dipar.Vn1_AVOM_ON(mdl_value := MODULE_UCP1_A2_DI3.VALUE.2, mdl_flt := MODULE_UCP1_A2_DI3.HwError); //Вентилятор АВОМД+Н+У №1 включен
dipar.Vn2_AVOM_ON(mdl_value := MODULE_UCP1_A2_DI3.VALUE.3, mdl_flt := MODULE_UCP1_A2_DI3.HwError); //Вентилятор АВОМД+Н+У №2 включен
dipar.VV_VOU_ON(mdl_value := MODULE_UCP1_A2_DI3.VALUE.4, mdl_flt := MODULE_UCP1_A2_DI3.HwError); //Вентилятор ВОУ включен
dipar.VVN_ON(mdl_value := MODULE_UCP1_A2_DI3.VALUE.5, mdl_flt := MODULE_UCP1_A2_DI3.HwError); //Вытяжной вентилятор нагнетателя ВВН включен
dipar.TRKready(mdl_value := MODULE_UCP1_A2_DI3.VALUE.8, mdl_flt := MODULE_UCP1_A2_DI3.HwError); //ТРК: готовность
dipar.TRKalr(mdl_value := MODULE_UCP1_A2_DI3.VALUE.9, mdl_flt := MODULE_UCP1_A2_DI3.HwError); //ТРК: авария
dipar.Ptg_inDG_Pn(mdl_value := MODULE_UCP1_A2_DI3.VALUE.17, mdl_flt := MODULE_UCP1_A2_DI3.HwError); //Давление газа перед дозатором газа Предупредительное
dipar.Vn3_AVOM_ON(mdl_value := MODULE_UCP1_A2_DI3.VALUE.21, mdl_flt := MODULE_UCP1_A2_DI3.HwError); //Вентилятор АВОМД+Н+У №3 включен
dipar.Vn4_AVOM_ON(mdl_value := MODULE_UCP1_A2_DI3.VALUE.22, mdl_flt := MODULE_UCP1_A2_DI3.HwError); //Вентилятор АВОМД+Н+У №4 включен
dipar.Ptg_inDG_An(mdl_value := MODULE_UCP1_A2_DI3.VALUE.23, mdl_flt := MODULE_UCP1_A2_DI3.HwError); //Давление газа перед дозатором газа Аварийное
dipar.Fuse_AO_UCP1(mdl_value := MODULE_UCP1_A2_DI4.VALUE.16, mdl_flt := MODULE_UCP1_A2_DI4.HwError); //диаг. Предохранитель UCP1-XTFU1:1 питания модулей AO исправен
dipar.Fuse_DO_UCP1(mdl_value := MODULE_UCP1_A2_DI4.VALUE.17, mdl_flt := MODULE_UCP1_A2_DI4.HwError); //диаг. Предохранитель UCP1-XTFU1:2 питания модулей DO исправен
dipar.Fuse_Air_UCP1(mdl_value := MODULE_UCP1_A2_DI4.VALUE.18, mdl_flt := MODULE_UCP1_A2_DI4.HwError); //диаг. Предохранитель UCP1--XTFU6:1 питания датчиков температуры и влажности
dipar.AO_PRU_1_ai(mdl_value := MODULE_UE1_A1_DI1.CH01.VALUE, mdl_flt := MODULE_UE1_A1_DI1.CH01.STATUS.0 OR MODULE_UE1_A1_DI1.HwError); //Кнопка АО на ПРУ сигнал 1 (НР)
dipar.AO_PRU_1(mdl_value := dipar.AO_PRU_1_ai.value, mdl_hwError := dipar.AO_PRU_1_ai.flt, mdl_sc := dipar.AO_PRU_1_ai.sc, mdl_brk := dipar.AO_PRU_1_ai.brk); //Кнопка АО на ПРУ сигнал 1 (НР)

dipar.Kr1_off_ai(mdl_value := MODULE_UE1_A1_DI1.CH02.VALUE, mdl_flt := MODULE_UE1_A1_DI1.CH02.STATUS.0 OR MODULE_UE1_A1_DI1.HwError); //Кран 1 закрыт
dipar.Kr1_off(mdl_value := dipar.Kr1_off_ai.value, mdl_hwError := dipar.Kr1_off_ai.flt, mdl_sc := dipar.Kr1_off_ai.sc, mdl_brk := dipar.Kr1_off_ai.brk); //Кран 1 закрыт

dipar.Kr2_off_ai(mdl_value := MODULE_UE1_A1_DI1.CH03.VALUE, mdl_flt := MODULE_UE1_A1_DI1.CH03.STATUS.0 OR MODULE_UE1_A1_DI1.HwError); //Кран 2 закрыт
dipar.Kr2_off(mdl_value := dipar.Kr2_off_ai.value, mdl_hwError := dipar.Kr2_off_ai.flt, mdl_sc := dipar.Kr2_off_ai.sc, mdl_brk := dipar.Kr2_off_ai.brk); //Кран 2 закрыт

dipar.Kr4_off_ai(mdl_value := MODULE_UE1_A1_DI1.CH04.VALUE, mdl_flt := MODULE_UE1_A1_DI1.CH04.STATUS.0 OR MODULE_UE1_A1_DI1.HwError); //Кран 4 закрыт
dipar.Kr4_off(mdl_value := dipar.Kr4_off_ai.value, mdl_hwError := dipar.Kr4_off_ai.flt, mdl_sc := dipar.Kr4_off_ai.sc, mdl_brk := dipar.Kr4_off_ai.brk); //Кран 4 закрыт

dipar.Kr5_off_ai(mdl_value := MODULE_UE1_A1_DI1.CH05.VALUE, mdl_flt := MODULE_UE1_A1_DI1.CH05.STATUS.0 OR MODULE_UE1_A1_DI1.HwError); //Кран 5 закрыт
dipar.Kr5_off(mdl_value := dipar.Kr5_off_ai.value, mdl_hwError := dipar.Kr5_off_ai.flt, mdl_sc := dipar.Kr5_off_ai.sc, mdl_brk := dipar.Kr5_off_ai.brk); //Кран 5 закрыт

dipar.Kr6_off_ai(mdl_value := MODULE_UE1_A1_DI1.CH06.VALUE, mdl_flt := MODULE_UE1_A1_DI1.CH06.STATUS.0 OR MODULE_UE1_A1_DI1.HwError); //Кран 6 закрыт
dipar.Kr6_off(mdl_value := dipar.Kr6_off_ai.value, mdl_hwError := dipar.Kr6_off_ai.flt, mdl_sc := dipar.Kr6_off_ai.sc, mdl_brk := dipar.Kr6_off_ai.brk); //Кран 6 закрыт

dipar.Kr12_off_ai(mdl_value := MODULE_UE1_A1_DI1.CH07.VALUE, mdl_flt := MODULE_UE1_A1_DI1.CH07.STATUS.0 OR MODULE_UE1_A1_DI1.HwError); //Кран 12 закрыт (т.г.)
dipar.Kr12_off(mdl_value := dipar.Kr12_off_ai.value, mdl_hwError := dipar.Kr12_off_ai.flt, mdl_sc := dipar.Kr12_off_ai.sc, mdl_brk := dipar.Kr12_off_ai.brk); //Кран 12 закрыт (т.г.)

dipar.Kr9_off_ai(mdl_value := MODULE_UE1_A1_DI1.CH08.VALUE, mdl_flt := MODULE_UE1_A1_DI1.CH08.STATUS.0 OR MODULE_UE1_A1_DI1.HwError); //Кран 9 закрыт (т.газ. свеча.)
dipar.Kr9_off(mdl_value := dipar.Kr9_off_ai.value, mdl_hwError := dipar.Kr9_off_ai.flt, mdl_sc := dipar.Kr9_off_ai.sc, mdl_brk := dipar.Kr9_off_ai.brk); //Кран 9 закрыт (т.газ. свеча.)

dipar.Kr11_off_ai(mdl_value := MODULE_UE1_A1_DI1.CH09.VALUE, mdl_flt := MODULE_UE1_A1_DI1.CH09.STATUS.0 OR MODULE_UE1_A1_DI1.HwError); //Кран 11 закрыт (п.г.)
dipar.Kr11_off(mdl_value := dipar.Kr11_off_ai.value, mdl_hwError := dipar.Kr11_off_ai.flt, mdl_sc := dipar.Kr11_off_ai.sc, mdl_brk := dipar.Kr11_off_ai.brk); //Кран 11 закрыт (п.г.)

dipar.Kr10_off_ai(mdl_value := MODULE_UE1_A1_DI1.CH10.VALUE, mdl_flt := MODULE_UE1_A1_DI1.CH10.STATUS.0 OR MODULE_UE1_A1_DI1.HwError); //Кран 10 закрыт (п.газ. свеча.)
dipar.Kr10_off(mdl_value := dipar.Kr10_off_ai.value, mdl_hwError := dipar.Kr10_off_ai.flt, mdl_sc := dipar.Kr10_off_ai.sc, mdl_brk := dipar.Kr10_off_ai.brk); //Кран 10 закрыт (п.газ. свеча.)

dipar.KPV1_off_ai(mdl_value := MODULE_UE1_A1_DI1.CH11.VALUE, mdl_flt := MODULE_UE1_A1_DI1.CH11.STATUS.0 OR MODULE_UE1_A1_DI1.HwError); //КПВ-1 закрыт
dipar.KPV1_off(mdl_value := dipar.KPV1_off_ai.value, mdl_hwError := dipar.KPV1_off_ai.flt, mdl_sc := dipar.KPV1_off_ai.sc, mdl_brk := dipar.KPV1_off_ai.brk); //КПВ-1 закрыт

dipar.KPV2_off_ai(mdl_value := MODULE_UE1_A1_DI1.CH12.VALUE, mdl_flt := MODULE_UE1_A1_DI1.CH12.STATUS.0 OR MODULE_UE1_A1_DI1.HwError); //КПВ-2 закрыт
dipar.KPV2_off(mdl_value := dipar.KPV2_off_ai.value, mdl_hwError := dipar.KPV2_off_ai.flt, mdl_sc := dipar.KPV2_off_ai.sc, mdl_brk := dipar.KPV2_off_ai.brk); //КПВ-2 закрыт

dipar.KPV3_off_ai(mdl_value := MODULE_UE1_A1_DI1.CH13.VALUE, mdl_flt := MODULE_UE1_A1_DI1.CH13.STATUS.0 OR MODULE_UE1_A1_DI1.HwError); //КПВ-3 закрыт
dipar.KPV3_off(mdl_value := dipar.KPV3_off_ai.value, mdl_hwError := dipar.KPV3_off_ai.flt, mdl_sc := dipar.KPV3_off_ai.sc, mdl_brk := dipar.KPV3_off_ai.brk); //КПВ-3 закрыт

dipar.KPV4_off_ai(mdl_value := MODULE_UE1_A1_DI1.CH14.VALUE, mdl_flt := MODULE_UE1_A1_DI1.CH14.STATUS.0 OR MODULE_UE1_A1_DI1.HwError); //КПВ-4 закрыт
dipar.KPV4_off(mdl_value := dipar.KPV4_off_ai.value, mdl_hwError := dipar.KPV4_off_ai.flt, mdl_sc := dipar.KPV4_off_ai.sc, mdl_brk := dipar.KPV4_off_ai.brk); //КПВ-4 закрыт

dipar.KPV5_off_ai(mdl_value := MODULE_UE1_A1_DI1.CH15.VALUE, mdl_flt := MODULE_UE1_A1_DI1.CH15.STATUS.0 OR MODULE_UE1_A1_DI1.HwError); //КПВ-5 закрыт
dipar.KPV5_off(mdl_value := dipar.KPV5_off_ai.value, mdl_hwError := dipar.KPV5_off_ai.flt, mdl_sc := dipar.KPV5_off_ai.sc, mdl_brk := dipar.KPV5_off_ai.brk); //КПВ-5 закрыт

dipar.SK_off_ai(mdl_value := MODULE_UE1_A1_DI1.CH16.VALUE, mdl_flt := MODULE_UE1_A1_DI1.CH16.STATUS.0 OR MODULE_UE1_A1_DI1.HwError); //СК закрыт
dipar.SK_off(mdl_value := dipar.SK_off_ai.value, mdl_hwError := dipar.SK_off_ai.flt, mdl_sc := dipar.SK_off_ai.sc, mdl_brk := dipar.SK_off_ai.brk); //СК закрыт

dipar.AO_PRU_2_ai(mdl_value := MODULE_UE1_A1_DI2.CH01.VALUE, mdl_flt := MODULE_UE1_A1_DI2.CH01.STATUS.0 OR MODULE_UE1_A1_DI2.HwError); //Кнопка АО на ПРУ сигнал 2 (НЗ)
dipar.AO_PRU_2(mdl_value := dipar.AO_PRU_2_ai.value, mdl_hwError := dipar.AO_PRU_2_ai.flt, mdl_sc := dipar.AO_PRU_2_ai.sc, mdl_brk := dipar.AO_PRU_2_ai.brk); //Кнопка АО на ПРУ сигнал 2 (НЗ)

dipar.Kr1_ON_ai(mdl_value := MODULE_UE1_A1_DI2.CH02.VALUE, mdl_flt := MODULE_UE1_A1_DI2.CH02.STATUS.0 OR MODULE_UE1_A1_DI2.HwError); //Кран 1 открыт
dipar.Kr1_ON(mdl_value := dipar.Kr1_ON_ai.value, mdl_hwError := dipar.Kr1_ON_ai.flt, mdl_sc := dipar.Kr1_ON_ai.sc, mdl_brk := dipar.Kr1_ON_ai.brk); //Кран 1 открыт

dipar.Kr2_ON_ai(mdl_value := MODULE_UE1_A1_DI2.CH03.VALUE, mdl_flt := MODULE_UE1_A1_DI2.CH03.STATUS.0 OR MODULE_UE1_A1_DI2.HwError); //Кран 2 открыт
dipar.Kr2_ON(mdl_value := dipar.Kr2_ON_ai.value, mdl_hwError := dipar.Kr2_ON_ai.flt, mdl_sc := dipar.Kr2_ON_ai.sc, mdl_brk := dipar.Kr2_ON_ai.brk); //Кран 2 открыт

dipar.Kr4_ON_ai(mdl_value := MODULE_UE1_A1_DI2.CH04.VALUE, mdl_flt := MODULE_UE1_A1_DI2.CH04.STATUS.0 OR MODULE_UE1_A1_DI2.HwError); //Кран 4 открыт
dipar.Kr4_ON(mdl_value := dipar.Kr4_ON_ai.value, mdl_hwError := dipar.Kr4_ON_ai.flt, mdl_sc := dipar.Kr4_ON_ai.sc, mdl_brk := dipar.Kr4_ON_ai.brk); //Кран 4 открыт

dipar.Kr5_ON_ai(mdl_value := MODULE_UE1_A1_DI2.CH05.VALUE, mdl_flt := MODULE_UE1_A1_DI2.CH05.STATUS.0 OR MODULE_UE1_A1_DI2.HwError); //Кран 5 открыт
dipar.Kr5_ON(mdl_value := dipar.Kr5_ON_ai.value, mdl_hwError := dipar.Kr5_ON_ai.flt, mdl_sc := dipar.Kr5_ON_ai.sc, mdl_brk := dipar.Kr5_ON_ai.brk); //Кран 5 открыт

dipar.Kr6_ON_ai(mdl_value := MODULE_UE1_A1_DI2.CH06.VALUE, mdl_flt := MODULE_UE1_A1_DI2.CH06.STATUS.0 OR MODULE_UE1_A1_DI2.HwError); //Кран 6 открыт
dipar.Kr6_ON(mdl_value := dipar.Kr6_ON_ai.value, mdl_hwError := dipar.Kr6_ON_ai.flt, mdl_sc := dipar.Kr6_ON_ai.sc, mdl_brk := dipar.Kr6_ON_ai.brk); //Кран 6 открыт

dipar.Kr12_ON_ai(mdl_value := MODULE_UE1_A1_DI2.CH07.VALUE, mdl_flt := MODULE_UE1_A1_DI2.CH07.STATUS.0 OR MODULE_UE1_A1_DI2.HwError); //Кран 12 открыт (т.г.)
dipar.Kr12_ON(mdl_value := dipar.Kr12_ON_ai.value, mdl_hwError := dipar.Kr12_ON_ai.flt, mdl_sc := dipar.Kr12_ON_ai.sc, mdl_brk := dipar.Kr12_ON_ai.brk); //Кран 12 открыт (т.г.)

dipar.Kr9_ON_ai(mdl_value := MODULE_UE1_A1_DI2.CH08.VALUE, mdl_flt := MODULE_UE1_A1_DI2.CH08.STATUS.0 OR MODULE_UE1_A1_DI2.HwError); //Кран 9 открыт (т.газ. свеча.)
dipar.Kr9_ON(mdl_value := dipar.Kr9_ON_ai.value, mdl_hwError := dipar.Kr9_ON_ai.flt, mdl_sc := dipar.Kr9_ON_ai.sc, mdl_brk := dipar.Kr9_ON_ai.brk); //Кран 9 открыт (т.газ. свеча.)

dipar.Kr11_ON_ai(mdl_value := MODULE_UE1_A1_DI2.CH09.VALUE, mdl_flt := MODULE_UE1_A1_DI2.CH09.STATUS.0 OR MODULE_UE1_A1_DI2.HwError); //Кран 11 открыт (п.г.)
dipar.Kr11_ON(mdl_value := dipar.Kr11_ON_ai.value, mdl_hwError := dipar.Kr11_ON_ai.flt, mdl_sc := dipar.Kr11_ON_ai.sc, mdl_brk := dipar.Kr11_ON_ai.brk); //Кран 11 открыт (п.г.)

dipar.Kr10_ON_ai(mdl_value := MODULE_UE1_A1_DI2.CH10.VALUE, mdl_flt := MODULE_UE1_A1_DI2.CH10.STATUS.0 OR MODULE_UE1_A1_DI2.HwError); //Кран 10 открыт (п.газ. свеча.)
dipar.Kr10_ON(mdl_value := dipar.Kr10_ON_ai.value, mdl_hwError := dipar.Kr10_ON_ai.flt, mdl_sc := dipar.Kr10_ON_ai.sc, mdl_brk := dipar.Kr10_ON_ai.brk); //Кран 10 открыт (п.газ. свеча.)

dipar.KPV1_ON_ai(mdl_value := MODULE_UE1_A1_DI2.CH11.VALUE, mdl_flt := MODULE_UE1_A1_DI2.CH11.STATUS.0 OR MODULE_UE1_A1_DI2.HwError); //КПВ-1 открыт
dipar.KPV1_ON(mdl_value := dipar.KPV1_ON_ai.value, mdl_hwError := dipar.KPV1_ON_ai.flt, mdl_sc := dipar.KPV1_ON_ai.sc, mdl_brk := dipar.KPV1_ON_ai.brk); //КПВ-1 открыт

dipar.KPV2_ON_ai(mdl_value := MODULE_UE1_A1_DI2.CH12.VALUE, mdl_flt := MODULE_UE1_A1_DI2.CH12.STATUS.0 OR MODULE_UE1_A1_DI2.HwError); //КПВ-2 открыт
dipar.KPV2_ON(mdl_value := dipar.KPV2_ON_ai.value, mdl_hwError := dipar.KPV2_ON_ai.flt, mdl_sc := dipar.KPV2_ON_ai.sc, mdl_brk := dipar.KPV2_ON_ai.brk); //КПВ-2 открыт

dipar.KPV3_ON_ai(mdl_value := MODULE_UE1_A1_DI2.CH13.VALUE, mdl_flt := MODULE_UE1_A1_DI2.CH13.STATUS.0 OR MODULE_UE1_A1_DI2.HwError); //КПВ-3 открыт
dipar.KPV3_ON(mdl_value := dipar.KPV3_ON_ai.value, mdl_hwError := dipar.KPV3_ON_ai.flt, mdl_sc := dipar.KPV3_ON_ai.sc, mdl_brk := dipar.KPV3_ON_ai.brk); //КПВ-3 открыт

dipar.KPV4_ON_ai(mdl_value := MODULE_UE1_A1_DI2.CH14.VALUE, mdl_flt := MODULE_UE1_A1_DI2.CH14.STATUS.0 OR MODULE_UE1_A1_DI2.HwError); //КПВ-4 открыт
dipar.KPV4_ON(mdl_value := dipar.KPV4_ON_ai.value, mdl_hwError := dipar.KPV4_ON_ai.flt, mdl_sc := dipar.KPV4_ON_ai.sc, mdl_brk := dipar.KPV4_ON_ai.brk); //КПВ-4 открыт

dipar.KPV5_ON_ai(mdl_value := MODULE_UE1_A1_DI2.CH15.VALUE, mdl_flt := MODULE_UE1_A1_DI2.CH15.STATUS.0 OR MODULE_UE1_A1_DI2.HwError); //КПВ-5 открыт
dipar.KPV5_ON(mdl_value := dipar.KPV5_ON_ai.value, mdl_hwError := dipar.KPV5_ON_ai.flt, mdl_sc := dipar.KPV5_ON_ai.sc, mdl_brk := dipar.KPV5_ON_ai.brk); //КПВ-5 открыт

dipar.SK_ON_ai(mdl_value := MODULE_UE1_A1_DI2.CH16.VALUE, mdl_flt := MODULE_UE1_A1_DI2.CH16.STATUS.0 OR MODULE_UE1_A1_DI2.HwError); //СК открыт
dipar.SK_ON(mdl_value := dipar.SK_ON_ai.value, mdl_hwError := dipar.SK_ON_ai.flt, mdl_sc := dipar.SK_ON_ai.sc, mdl_brk := dipar.SK_ON_ai.brk); //СК открыт

dipar.PNS_ON_ai(mdl_value := MODULE_UE1_A1_DI3.CH01.VALUE, mdl_flt := MODULE_UE1_A1_DI3.CH01.STATUS.0 OR MODULE_UE1_A1_DI3.HwError); //Пусковой насос смазки включен
dipar.PNS_ON(mdl_value := dipar.PNS_ON_ai.value, mdl_hwError := dipar.PNS_ON_ai.flt, mdl_sc := dipar.PNS_ON_ai.sc, mdl_brk := dipar.PNS_ON_ai.brk); //Пусковой насос смазки включен

dipar.PNU_ON_ai(mdl_value := MODULE_UE1_A1_DI3.CH02.VALUE, mdl_flt := MODULE_UE1_A1_DI3.CH02.STATUS.0 OR MODULE_UE1_A1_DI3.HwError); //Пусковой насос уплотнения включен
dipar.PNU_ON(mdl_value := dipar.PNU_ON_ai.value, mdl_hwError := dipar.PNU_ON_ai.flt, mdl_sc := dipar.PNU_ON_ai.sc, mdl_brk := dipar.PNU_ON_ai.brk); //Пусковой насос уплотнения включен

dipar.Vs_D_Pv(mdl_value := MODULE_UE1_A1_DI4.VALUE.8, mdl_flt := MODULE_UE1_A1_DI4.HwError); //Повышенная вибрация двигателя
dipar.Vs_D_Av(mdl_value := MODULE_UE1_A1_DI4.VALUE.9, mdl_flt := MODULE_UE1_A1_DI4.HwError); //Опасная вибрация двигателя
dipar.Zs_Nl(mdl_value := MODULE_UE1_A1_DI4.VALUE.17, mdl_flt := MODULE_UE1_A1_DI4.HwError); //Осевой сдвиг ротора Н Аварийный
dipar.Pg_outKR1(mdl_value := MODULE_UE1_A1_DI4.VALUE.19, mdl_flt := MODULE_UE1_A1_DI4.HwError); //Давление газа после крана 1
dipar.Pm_N_Pn(mdl_value := MODULE_UE1_A1_DI4.VALUE.22, mdl_flt := MODULE_UE1_A1_DI4.HwError); //Давление масла смазки Н предупредительная
dipar.Exh_VOU(mdl_value := MODULE_UE1_A1_DI4.VALUE.23, mdl_flt := MODULE_UE1_A1_DI4.HwError); //Разрежение в ВОУ
dipar.Pg_InKR13(mdl_value := MODULE_UE1_A1_DI4.VALUE.24, mdl_flt := MODULE_UE1_A1_DI4.HwError); //Давление газа до крана 13 (воздушного стартера)
dipar.Pm_Starter_Av(mdl_value := MODULE_UE1_A1_DI4.VALUE.25, mdl_flt := MODULE_UE1_A1_DI4.HwError); //Давление масла смазки воздушного стартера высокий уровень
dipar.Pm_Starter_An(mdl_value := MODULE_UE1_A1_DI4.VALUE.26, mdl_flt := MODULE_UE1_A1_DI4.HwError); //Давление масла смазки воздушного стартера низкий уровень
dipar.EAO_PRU_1(mdl_value := MODULE_UE1_A1_DI4.VALUE.28, mdl_flt := MODULE_UE1_A1_DI4.HwError); //Кнопка ЭАО на ПРУ нажата сигнал 1 (НР)
dipar.EAO_PRU_2(mdl_value := MODULE_UE1_A1_DI4.VALUE.29, mdl_flt := MODULE_UE1_A1_DI4.HwError); //Кнопка ЭАО на ПРУ нажата сигнал 2 (НЗ)
dipar.EAO_PRU_3(mdl_value := MODULE_UE1_A1_DI4.VALUE.30, mdl_flt := MODULE_UE1_A1_DI4.HwError); //Кнопка ЭАО на ПРУ нажата сигнал 3 (НЗ)
dipar.BEAO(mdl_value := MODULE_UE1_A1_DI4.VALUE.31, mdl_flt := MODULE_UE1_A1_DI4.HwError); //БЭАО сработал
dipar.Kr13_ON(mdl_value := MODULE_UE1_A1_DI5.VALUE.0, mdl_flt := MODULE_UE1_A1_DI5.HwError); //Заслонка ВC (кран 13) открыта
dipar.BZA_alr(mdl_value := MODULE_UE1_A1_DI5.VALUE.1, mdl_flt := MODULE_UE1_A1_DI5.HwError); //БЗА. Авария
dipar.BZA_ready_1(mdl_value := MODULE_UE1_A1_DI5.VALUE.2, mdl_flt := MODULE_UE1_A1_DI5.HwError); //БЗА. Готовность 1
dipar.BZA_ready_2(mdl_value := MODULE_UE1_A1_DI5.VALUE.3, mdl_flt := MODULE_UE1_A1_DI5.HwError); //БЗА. Готовность 2
dipar.U_CC_cntrl(mdl_value := MODULE_UE1_A1_DI5.VALUE.24, mdl_flt := MODULE_UE1_A1_DI5.HwError); //Контроль питания СС
dipar.Chip_outD(mdl_value := MODULE_UE1_A1_DI5.VALUE.25, mdl_flt := MODULE_UE1_A1_DI5.HwError); //Стружка в масле на выходе Д
dipar.Ace_alr(mdl_value := MODULE_UE1_A1_DI5.VALUE.26, mdl_flt := MODULE_UE1_A1_DI5.HwError); //Сигнализатор обледенения
dipar.kcdo_Kr1_off(mdl_value := MODULE_UE1_A1_DI6.VALUE.0, mdl_flt := MODULE_UE1_A1_DI6.HwError); //диаг. Кран 1 закрыть
dipar.kcdo_Kr1m_ON(mdl_value := MODULE_UE1_A1_DI6.VALUE.1, mdl_flt := MODULE_UE1_A1_DI6.HwError); //диаг. Кран 1 смазка
dipar.kcdo_Kr2_off(mdl_value := MODULE_UE1_A1_DI6.VALUE.2, mdl_flt := MODULE_UE1_A1_DI6.HwError); //диаг. Кран 2 закрыть
dipar.kcdo_Kr2m_ON(mdl_value := MODULE_UE1_A1_DI6.VALUE.3, mdl_flt := MODULE_UE1_A1_DI6.HwError); //диаг. Кран 2 смазка
dipar.kcdo_Kr4_off(mdl_value := MODULE_UE1_A1_DI6.VALUE.4, mdl_flt := MODULE_UE1_A1_DI6.HwError); //диаг. Кран 4 закрыть
dipar.kcdo_Kr4m_ON(mdl_value := MODULE_UE1_A1_DI6.VALUE.5, mdl_flt := MODULE_UE1_A1_DI6.HwError); //диаг. Кран 4 смазка
dipar.kcdo_Kr5_ON(mdl_value := MODULE_UE1_A1_DI6.VALUE.6, mdl_flt := MODULE_UE1_A1_DI6.HwError); //диаг. Кран 5 открыть
dipar.kcdo_Kr5m_ON(mdl_value := MODULE_UE1_A1_DI6.VALUE.7, mdl_flt := MODULE_UE1_A1_DI6.HwError); //диаг. Кран 5 смазка
dipar.kcdo_Kr6_off(mdl_value := MODULE_UE1_A1_DI6.VALUE.8, mdl_flt := MODULE_UE1_A1_DI6.HwError); //диаг. Кран 6 закрыть
dipar.kcdo_Kr6m_ON(mdl_value := MODULE_UE1_A1_DI6.VALUE.9, mdl_flt := MODULE_UE1_A1_DI6.HwError); //диаг. Кран 6 смазка
dipar.kcdo_KR12_off(mdl_value := MODULE_UE1_A1_DI6.VALUE.10, mdl_flt := MODULE_UE1_A1_DI6.HwError); //диаг. Кран 12 закрыть (т.г.)
dipar.kcdo_KR12m_ON(mdl_value := MODULE_UE1_A1_DI6.VALUE.11, mdl_flt := MODULE_UE1_A1_DI6.HwError); //диаг. Кран 12 смазка
dipar.kcdo_KR9m_ON(mdl_value := MODULE_UE1_A1_DI6.VALUE.13, mdl_flt := MODULE_UE1_A1_DI6.HwError); //диаг. Кран 9 смазка
dipar.kcdo_Kr11_ON(mdl_value := MODULE_UE1_A1_DI6.VALUE.14, mdl_flt := MODULE_UE1_A1_DI6.HwError); //диаг. Кран 11 открыть (п.г.)
dipar.kcdo_Kr11m_ON(mdl_value := MODULE_UE1_A1_DI6.VALUE.15, mdl_flt := MODULE_UE1_A1_DI6.HwError); //диаг. Кран 11 смазка
dipar.kcdo_Kr10m_ON(mdl_value := MODULE_UE1_A1_DI6.VALUE.17, mdl_flt := MODULE_UE1_A1_DI6.HwError); //диаг. Кран 10 смазка
dipar.kcdo_KPV15_ON(mdl_value := MODULE_UE1_A1_DI6.VALUE.18, mdl_flt := MODULE_UE1_A1_DI6.HwError); //диаг. Включение КПВ 1,5
dipar.kcdo_KPV23_off(mdl_value := MODULE_UE1_A1_DI6.VALUE.19, mdl_flt := MODULE_UE1_A1_DI6.HwError); //диаг. Включение КПВ 2,3
dipar.kcdo_KPV4_off(mdl_value := MODULE_UE1_A1_DI6.VALUE.20, mdl_flt := MODULE_UE1_A1_DI6.HwError); //диаг. Включение КПВ 4
dipar.kcdo_SK_ON(mdl_value := MODULE_UE1_A1_DI6.VALUE.21, mdl_flt := MODULE_UE1_A1_DI6.HwError); //диаг. Стопорный клапан открыть
dipar.kcdo_Kr1_ON(mdl_value := MODULE_UE1_A1_DI7.VALUE.0, mdl_flt := MODULE_UE1_A1_DI7.HwError); //диаг. Кран 1 открыть
dipar.kcdo_Kr2_ON(mdl_value := MODULE_UE1_A1_DI7.VALUE.1, mdl_flt := MODULE_UE1_A1_DI7.HwError); //диаг. Кран 2 открыть
dipar.kcdo_Kr4_ON(mdl_value := MODULE_UE1_A1_DI7.VALUE.2, mdl_flt := MODULE_UE1_A1_DI7.HwError); //диаг. Кран 4 открыть
dipar.kcdo_Kr5_off(mdl_value := MODULE_UE1_A1_DI7.VALUE.3, mdl_flt := MODULE_UE1_A1_DI7.HwError); //диаг. Кран 5 закрыть
dipar.kcdo_Kr6_ON(mdl_value := MODULE_UE1_A1_DI7.VALUE.4, mdl_flt := MODULE_UE1_A1_DI7.HwError); //диаг. Кран 6 открыть
dipar.kcdo_Kr12_ON(mdl_value := MODULE_UE1_A1_DI7.VALUE.5, mdl_flt := MODULE_UE1_A1_DI7.HwError); //диаг. Кран 12 открыть (т.г.)
dipar.kcdo_Kr11_off(mdl_value := MODULE_UE1_A1_DI7.VALUE.7, mdl_flt := MODULE_UE1_A1_DI7.HwError); //диаг. Кран 11 закрыть (п.г.)
dipar.kcdo_Sound_ON(mdl_value := MODULE_UE1_A1_DI7.VALUE.10, mdl_flt := MODULE_UE1_A1_DI7.HwError); //диаг. ЗВУКОВУЮ СИГНАЛИЗАЦИЮ в ГЩУ ВКЛЮЧИТЬ
dipar.kcdo_VNA_ON(mdl_value := MODULE_UE1_A1_DI7.VALUE.15, mdl_flt := MODULE_UE1_A1_DI7.HwError); //диаг. Эл. магнит управления ВНА включить
dipar.Fuse_DO_UE1(mdl_value := MODULE_UE1_A1_DI7.VALUE.16, mdl_flt := MODULE_UE1_A1_DI7.HwError); //диаг. Предохранитель UE1-XTFU1:2 питания модулей DO исправен
dipar.EV1(mdl_value := MODULE_UPD1_A1_DI1.VALUE.0, mdl_flt := MODULE_UPD1_A1_DI1.HwError); //Перегрузка фильтра EV1 (Осн.)
dipar.EV2(mdl_value := MODULE_UPD1_A1_DI1.VALUE.1, mdl_flt := MODULE_UPD1_A1_DI1.HwError); //Перегрузка фильтра EV2 (Рез.)
dipar.AG1(mdl_value := MODULE_UPD1_A1_DI1.VALUE.2, mdl_flt := MODULE_UPD1_A1_DI1.HwError); //Контроль -AG1
dipar.AG2(mdl_value := MODULE_UPD1_A1_DI1.VALUE.3, mdl_flt := MODULE_UPD1_A1_DI1.HwError); //Контроль -AG2
dipar.AG5(mdl_value := MODULE_UPD1_A1_DI1.VALUE.4, mdl_flt := MODULE_UPD1_A1_DI1.HwError); //Контроль -AG5
dipar.AG6(mdl_value := MODULE_UPD1_A1_DI1.VALUE.5, mdl_flt := MODULE_UPD1_A1_DI1.HwError); //Контроль -AG6
dipar.AG8(mdl_value := MODULE_UPD1_A1_DI1.VALUE.6, mdl_flt := MODULE_UPD1_A1_DI1.HwError); //Контроль -AG8
dipar.AG9(mdl_value := MODULE_UPD1_A1_DI1.VALUE.7, mdl_flt := MODULE_UPD1_A1_DI1.HwError); //Контроль -AG9
dipar.AG10(mdl_value := MODULE_UPD1_A1_DI1.VALUE.8, mdl_flt := MODULE_UPD1_A1_DI1.HwError); //Контроль -AG10
dipar.AG15(mdl_value := MODULE_UPD1_A1_DI1.VALUE.9, mdl_flt := MODULE_UPD1_A1_DI1.HwError); //Контроль -AG15
dipar.AG16(mdl_value := MODULE_UPD1_A1_DI1.VALUE.10, mdl_flt := MODULE_UPD1_A1_DI1.HwError); //Контроль -AG16
dipar.AG17(mdl_value := MODULE_UPD1_A1_DI1.VALUE.11, mdl_flt := MODULE_UPD1_A1_DI1.HwError); //Контроль -AG17
dipar.AG18(mdl_value := MODULE_UPD1_A1_DI1.VALUE.12, mdl_flt := MODULE_UPD1_A1_DI1.HwError); //Контроль -AG18
dipar.Err_AUO1(mdl_value := MODULE_UPD1_A1_DI1.VALUE.13, mdl_flt := MODULE_UPD1_A1_DI1.HwError); //Ошибка -AUO1
dipar.U_main(mdl_value := MODULE_UPD1_A1_DI2.VALUE.0, mdl_flt := MODULE_UPD1_A1_DI2.HwError); //Контроль основного ввода питания (-KV1)
dipar.U_res(mdl_value := MODULE_UPD1_A1_DI2.VALUE.1, mdl_flt := MODULE_UPD1_A1_DI2.HwError); //Контроль резервного ввода питания (-KV2)
dipar.U_G_PLC(mdl_value := MODULE_UPD1_A1_DI2.VALUE.2, mdl_flt := MODULE_UPD1_A1_DI2.HwError); //Контроль замыкания на землю питания PLC
dipar.U_G_AI(mdl_value := MODULE_UPD1_A1_DI2.VALUE.3, mdl_flt := MODULE_UPD1_A1_DI2.HwError); //Контроль замыкания на землю питания AI
dipar.U_G_DI(mdl_value := MODULE_UPD1_A1_DI2.VALUE.4, mdl_flt := MODULE_UPD1_A1_DI2.HwError); //Контроль замыкания на землю питания DI
dipar.U_G_BIZ(mdl_value := MODULE_UPD1_A1_DI2.VALUE.5, mdl_flt := MODULE_UPD1_A1_DI2.HwError); //Контроль замыкания на FE питания БИЗ
dipar.U_G_AM(mdl_value := MODULE_UPD1_A1_DI2.VALUE.6, mdl_flt := MODULE_UPD1_A1_DI2.HwError); //Контроль замыкания на землю питания ИМ
dipar.U_AI(mdl_value := MODULE_UPD1_A1_DI2.VALUE.7, mdl_flt := MODULE_UPD1_A1_DI2.HwError); //Контроль питания AI
dipar.U_DI(mdl_value := MODULE_UPD1_A1_DI2.VALUE.8, mdl_flt := MODULE_UPD1_A1_DI2.HwError); //Контроль питания DI
dipar.U_BIZ(mdl_value := MODULE_UPD1_A1_DI2.VALUE.9, mdl_flt := MODULE_UPD1_A1_DI2.HwError); //Контроль питания БИЗ
dipar.U_AM(mdl_value := MODULE_UPD1_A1_DI2.VALUE.10, mdl_flt := MODULE_UPD1_A1_DI2.HwError); //Контроль питания ИМ
dipar.Uvs_24(mdl_value := MODULE_UPD1_A1_DI2.VALUE.11, mdl_flt := MODULE_UPD1_A1_DI2.HwError); //Контроль питания аппаратуры вибрации, =24 В
dipar.Uother_24(mdl_value := MODULE_UPD1_A1_DI2.VALUE.12, mdl_flt := MODULE_UPD1_A1_DI2.HwError); //Контроль питания дополнительного оборудования, =24В
dipar.U_AM2(mdl_value := MODULE_UPD1_A1_DI2.VALUE.13, mdl_flt := MODULE_UPD1_A1_DI2.HwError); //Контроль питания ИМ2
dipar.Utrk_res(mdl_value := MODULE_UPD1_A1_DI2.VALUE.14, mdl_flt := MODULE_UPD1_A1_DI2.HwError); //Контроль питания ТРК рез.
dipar.U_PRU(mdl_value := MODULE_UPD1_A1_DI2.VALUE.15, mdl_flt := MODULE_UPD1_A1_DI2.HwError); //Контроль питания ПРУ
dipar.AG3(mdl_value := MODULE_UPD1_A1_DI3.VALUE.0, mdl_flt := MODULE_UPD1_A1_DI3.HwError); //Контроль -AG3
dipar.AG4(mdl_value := MODULE_UPD1_A1_DI3.VALUE.1, mdl_flt := MODULE_UPD1_A1_DI3.HwError); //Контроль -AG4
dipar.Utrk_main(mdl_value := MODULE_UPD1_A1_DI3.VALUE.2, mdl_flt := MODULE_UPD1_A1_DI3.HwError); //Контроль питания ТРК осн.
dipar.EV3(mdl_value := MODULE_UPD1_A1_DI3.VALUE.4, mdl_flt := MODULE_UPD1_A1_DI3.HwError); //БЭО. Перегрузка фильтра EV3 (Осн. БЭО)
dipar.EV4(mdl_value := MODULE_UPD1_A1_DI3.VALUE.5, mdl_flt := MODULE_UPD1_A1_DI3.HwError); //БЭО. Перегрузка фильтра EV4 (Рез. БЭО)
dipar.Ubeo_main(mdl_value := MODULE_UPD1_A1_DI3.VALUE.6, mdl_flt := MODULE_UPD1_A1_DI3.HwError); //БЭО. Контроль основного ввода питания БЭО (-KV3)
dipar.Ubeo_res(mdl_value := MODULE_UPD1_A1_DI3.VALUE.7, mdl_flt := MODULE_UPD1_A1_DI3.HwError); //БЭО. Контроль резервного ввода питания БЭО (-KV4)
dipar.AG11(mdl_value := MODULE_UPD1_A1_DI3.VALUE.8, mdl_flt := MODULE_UPD1_A1_DI3.HwError); //БЭО. Контроль -AG11
dipar.AG12(mdl_value := MODULE_UPD1_A1_DI3.VALUE.9, mdl_flt := MODULE_UPD1_A1_DI3.HwError); //БЭО. Контроль -AG12
dipar.U_G_KR5(mdl_value := MODULE_UPD1_A1_DI3.VALUE.10, mdl_flt := MODULE_UPD1_A1_DI3.HwError); //БЭО. Контроль замыкания на землю питания БЭО (-KR5)
dipar.U_KEAO(mdl_value := MODULE_UPD1_A1_DI3.VALUE.11, mdl_flt := MODULE_UPD1_A1_DI3.HwError); //БЭО. Контроль питания кн. ЭАО
dipar.U_BEO(mdl_value := MODULE_UPD1_A1_DI3.VALUE.12, mdl_flt := MODULE_UPD1_A1_DI3.HwError); //БЭО. Контроль питания БЭО
dipar.U_BZA(mdl_value := MODULE_UPD1_A1_DI3.VALUE.13, mdl_flt := MODULE_UPD1_A1_DI3.HwError); //БЭО. Контроль питания БЗА

                  
END_FUNCTION

{region INFO}
(*
 Назначение: Используется для обработки выходных дискретных параметров
 Автор:      /Andrey/ 16.07.2025 17:15:05
 Версия ТЭ5: v00.00.01
 Проект:     KA107
*)
{endregion}
FUNCTION dopar_update : BOOL
VAR_INPUT
END_VAR
VAR
END_VAR

                    dopar.VV_VOU_ON(mdl_hwError := MODULE_UCP1_A2_DO1.HwError, mdl_value => MODULE_UCP1_A2_DO1.VALUE.16); //Включить вытяжной Вент.ВОУ
dopar.VV_VOU_OFF(mdl_hwError := MODULE_UCP1_A2_DO1.HwError, mdl_value => MODULE_UCP1_A2_DO1.VALUE.17); //Отключить вытяжной Вент.ВОУ
dopar.Vn1_AVOM_ON(mdl_hwError := MODULE_UCP1_A2_DO1.HwError, mdl_value => MODULE_UCP1_A2_DO1.VALUE.18); //Вентилятор 1 маслоохладителей АВОМ включить
dopar.Vn1_AVOM_OFF(mdl_hwError := MODULE_UCP1_A2_DO1.HwError, mdl_value => MODULE_UCP1_A2_DO1.VALUE.19); //Вентилятор 1 маслоохладителей АВОМ отключить
dopar.Vn2_AVOM_ON(mdl_hwError := MODULE_UCP1_A2_DO1.HwError, mdl_value => MODULE_UCP1_A2_DO1.VALUE.20); //Вентилятор 2 маслоохладителей АВОМ включить
dopar.Vn2_AVOM_OFF(mdl_hwError := MODULE_UCP1_A2_DO1.HwError, mdl_value => MODULE_UCP1_A2_DO1.VALUE.21); //Вентилятор 2 маслоохладителей АВОМ отключить
dopar.Vn3_AVOM_ON(mdl_hwError := MODULE_UCP1_A2_DO1.HwError, mdl_value => MODULE_UCP1_A2_DO1.VALUE.22); //Вентилятор 3 маслоохладителей АВОМ включить
dopar.Vn3_AVOM_OFF(mdl_hwError := MODULE_UCP1_A2_DO1.HwError, mdl_value => MODULE_UCP1_A2_DO1.VALUE.23); //Вентилятор 3 маслоохладителей АВОМ отключить
dopar.Vn4_AVOM_ON(mdl_hwError := MODULE_UCP1_A2_DO1.HwError, mdl_value => MODULE_UCP1_A2_DO1.VALUE.24); //Вентилятор 4 маслоохладителей АВОМ включить
dopar.Vn4_AVOM_OFF(mdl_hwError := MODULE_UCP1_A2_DO1.HwError, mdl_value => MODULE_UCP1_A2_DO1.VALUE.25); //Вентилятор 4 маслоохладителей АВОМ отключить
dopar.VVN_ON(mdl_hwError := MODULE_UCP1_A2_DO1.HwError, mdl_value => MODULE_UCP1_A2_DO1.VALUE.26); //Вытяжной вентилятор нагнетателя ВВН включить
dopar.VVN_OFF(mdl_hwError := MODULE_UCP1_A2_DO1.HwError, mdl_value => MODULE_UCP1_A2_DO1.VALUE.27); //Вытяжной вентилятор нагнетателя ВВН отключить
dopar.PNU_OFF(mdl_hwError := MODULE_UCP1_A2_DO1.HwError, mdl_value => MODULE_UCP1_A2_DO1.VALUE.30); //Пусковой насос уплотнения отключить
dopar.PNS_OFF(mdl_hwError := MODULE_UCP1_A2_DO1.HwError, mdl_value => MODULE_UCP1_A2_DO1.VALUE.31); //Пусковой насос смазки отключить
dopar.Kr1_OFF(kc_di := dipar.kcdo_Kr1_OFF.value, mdl_hwError := MODULE_UE1_A1_DO1.HwError, mdl_value => MODULE_UE1_A1_DO1.VALUE.0); //Кран 1 закрыть
dopar.Kr1m_ON(kc_di := dipar.kcdo_Kr1m_ON.value, mdl_hwError := MODULE_UE1_A1_DO1.HwError, mdl_value => MODULE_UE1_A1_DO1.VALUE.1); //Кран 1 смазка
dopar.Kr2_OFF(kc_di := dipar.kcdo_Kr2_OFF.value, mdl_hwError := MODULE_UE1_A1_DO1.HwError, mdl_value => MODULE_UE1_A1_DO1.VALUE.2); //Кран 2 закрыть
dopar.Kr2m_ON(kc_di := dipar.kcdo_Kr2m_ON.value, mdl_hwError := MODULE_UE1_A1_DO1.HwError, mdl_value => MODULE_UE1_A1_DO1.VALUE.3); //Кран 2 смазка
dopar.Kr4_OFF(kc_di := dipar.kcdo_Kr4_OFF.value, mdl_hwError := MODULE_UE1_A1_DO1.HwError, mdl_value => MODULE_UE1_A1_DO1.VALUE.4); //Кран 4 закрыть
dopar.Kr5_ON(kc_di := dipar.kcdo_Kr5_ON.value, mdl_hwError := MODULE_UE1_A1_DO1.HwError, mdl_value => MODULE_UE1_A1_DO1.VALUE.6); //Кран 5 открыть
dopar.Kr6_OFF(kc_di := dipar.kcdo_Kr6_OFF.value, mdl_hwError := MODULE_UE1_A1_DO1.HwError, mdl_value => MODULE_UE1_A1_DO1.VALUE.8); //Кран 6 закрыть
dopar.Kr6m_ON(kc_di := dipar.kcdo_Kr6m_ON.value, mdl_hwError := MODULE_UE1_A1_DO1.HwError, mdl_value => MODULE_UE1_A1_DO1.VALUE.9); //Кран 6 смазка
dopar.KR12_OFF(kc_di := dipar.kcdo_KR12_OFF.value, mdl_hwError := MODULE_UE1_A1_DO1.HwError, mdl_value => MODULE_UE1_A1_DO1.VALUE.10); //Кран 12 закрыть (т.г.), кран 9 (т.г. свеч.) открыть
dopar.Kr11_ON(kc_di := dipar.kcdo_Kr11_ON.value, mdl_hwError := MODULE_UE1_A1_DO1.HwError, mdl_value => MODULE_UE1_A1_DO1.VALUE.14); //Кран 11 открыть (п.г.) кран 10(п.г.свеч.) закрыть
dopar.KPV15_ON(kc_di := dipar.kcdo_KPV15_ON.value, mdl_hwError := MODULE_UE1_A1_DO1.HwError, mdl_value => MODULE_UE1_A1_DO1.VALUE.18); //Включение КПВ 1,5
dopar.KPV23_OFF(kc_di := dipar.kcdo_KPV23_OFF.value, mdl_hwError := MODULE_UE1_A1_DO1.HwError, mdl_value => MODULE_UE1_A1_DO1.VALUE.19); //Включение КПВ 2,3
dopar.KPV4_OFF(kc_di := dipar.kcdo_KPV4_OFF.value, mdl_hwError := MODULE_UE1_A1_DO1.HwError, mdl_value => MODULE_UE1_A1_DO1.VALUE.20); //Включение КПВ 4
dopar.SK_ON(kc_di := dipar.kcdo_SK_ON.value, mdl_hwError := MODULE_UE1_A1_DO1.HwError, mdl_value => MODULE_UE1_A1_DO1.VALUE.21); //Стопорный клапан открыть
dopar.PNS_ON(mdl_hwError := MODULE_UE1_A1_DO1.HwError, mdl_value => MODULE_UE1_A1_DO1.VALUE.29); //Пусковой насос смазки включить
dopar.PNU_ON(mdl_hwError := MODULE_UE1_A1_DO1.HwError, mdl_value => MODULE_UE1_A1_DO1.VALUE.30); //Пусковой насос уплотнения включить
dopar.BEO_w1(mdl_hwError := MODULE_UE1_A1_DO1.HwError, mdl_value => MODULE_UE1_A1_DO1.VALUE.31); //БЭО. Работа-1
dopar.Kr1_ON(kc_di := dipar.kcdo_Kr1_ON.value, mdl_hwError := MODULE_UE1_A1_DO2.HwError, mdl_value => MODULE_UE1_A1_DO2.VALUE.0); //Кран 1 открыть
dopar.Kr2_ON(kc_di := dipar.kcdo_Kr2_ON.value, mdl_hwError := MODULE_UE1_A1_DO2.HwError, mdl_value => MODULE_UE1_A1_DO2.VALUE.1); //Кран 2 открыть
dopar.Kr4_ON(kc_di := dipar.kcdo_Kr4_ON.value, mdl_hwError := MODULE_UE1_A1_DO2.HwError, mdl_value => MODULE_UE1_A1_DO2.VALUE.2); //Кран 4 открыть
dopar.Kr5_OFF(kc_di := dipar.kcdo_Kr5_OFF.value, mdl_hwError := MODULE_UE1_A1_DO2.HwError, mdl_value => MODULE_UE1_A1_DO2.VALUE.3); //Кран 5 закрыть
dopar.Kr6_ON(kc_di := dipar.kcdo_Kr6_ON.value, mdl_hwError := MODULE_UE1_A1_DO2.HwError, mdl_value => MODULE_UE1_A1_DO2.VALUE.4); //Кран 6 открыть
dopar.Kr12_ON(kc_di := dipar.kcdo_Kr12_ON.value, mdl_hwError := MODULE_UE1_A1_DO2.HwError, mdl_value => MODULE_UE1_A1_DO2.VALUE.5); //Кран 12 открыть (т.г.), кран 9 (т.г. свеч.) закрыть
dopar.Kr11_OFF(kc_di := dipar.kcdo_Kr11_OFF.value, mdl_hwError := MODULE_UE1_A1_DO2.HwError, mdl_value => MODULE_UE1_A1_DO2.VALUE.7); //Кран 11 закрыть (п.г.) Кран 10(п.г.свеч.) открыть
dopar.Sound_ON(kc_di := dipar.kcdo_Sound_ON.value, mdl_hwError := MODULE_UE1_A1_DO2.HwError, mdl_value => MODULE_UE1_A1_DO2.VALUE.10); //ЗВУКОВУЮ СИГНАЛИЗАЦИЮ в ГЩУ ВКЛЮЧИТЬ
dopar.VNA_ON(kc_di := dipar.kcdo_VNA_ON.value, mdl_hwError := MODULE_UE1_A1_DO2.HwError, mdl_value => MODULE_UE1_A1_DO2.VALUE.15); //Эл. магнит управления ВНА включить
dopar.AZ_ON(mdl_hwError := MODULE_UE1_A1_DO2.HwError, mdl_value => MODULE_UE1_A1_DO2.VALUE.17); //Включить агрегат зажигания
dopar.VNA_heat_ON(mdl_hwError := MODULE_UE1_A1_DO2.HwError, mdl_value => MODULE_UE1_A1_DO2.VALUE.18); //Обогрев ВНА включить
dopar.Kr13_ON(mdl_hwError := MODULE_UE1_A1_DO2.HwError, mdl_value => MODULE_UE1_A1_DO2.VALUE.21); //Кран 13 открыть (заслонка возд. стартера)
dopar.Kr15_ON(mdl_hwError := MODULE_UE1_A1_DO2.HwError, mdl_value => MODULE_UE1_A1_DO2.VALUE.22); //Кран 15 открыть
dopar.Vibr_ctrl(mdl_hwError := MODULE_UE1_A1_DO2.HwError, mdl_value => MODULE_UE1_A1_DO2.VALUE.28); //Контроль ИВ-Д-ПФ-1М.3Н.1-01
dopar.BZA_ctrl(mdl_hwError := MODULE_UE1_A1_DO2.HwError, mdl_value => MODULE_UE1_A1_DO2.VALUE.29); //Контроль БЗА
dopar.BZA_reset(mdl_hwError := MODULE_UE1_A1_DO2.HwError, mdl_value => MODULE_UE1_A1_DO2.VALUE.30); //Сброс БЗА
dopar.BEO_w2(mdl_hwError := MODULE_UE1_A1_DO2.HwError, mdl_value => MODULE_UE1_A1_DO2.VALUE.31); //БЭО. Работа-2

                  
END_FUNCTION

{region INFO}
(*
 Назначение: вызов функциональных блоков последовательностей подсистемы "Блок двигателя"
 Автор: /Разработчик/ 08.08.2025 9:04:03
 Версия: v00.00.18
 Проект: KA107
*)
{endregion}
FUNCTION bd_update : BOOL
VAR_INPUT
	cycle : REAL; //цикл вызова
END_VAR

                    //Пуск двигателя
Start_D(cycle := cycle);

                  
END_FUNCTION

{region INFO}
(*
 Наименование последовательности: Пуск двигателя
 Автор: /Разработчик/ 08.08.2025 9:04:03
 Версия: v00.00.18
 Проект: KA107
*)
{endregion}
{attribute 'symbol' := 'none'}
FUNCTION_BLOCK PUBLIC T_Start_D
VAR_INPUT
	cycle : REAL; //цикл вызова
END_VAR
VAR_OUTPUT
	cmd_KR11_On : BOOL; //Открытие крана 11, закрытие крана 10
	check_Ntk : BOOL; //Проверка Nтк
	cmd_KR12_On : BOOL; //Открытие крана 12, закрытие крана 9
	cmd_VNA_On : BOOL; //Включение Э/М ВНА
	cmd_KPV_On : BOOL; //Открыть КПВ
	cmd_VS_On : BOOL; //Пуск воздушного стартера
	cmd_sh_TG_On : BOOL; //Взвести защиту по ТГ
	cmd_SK_On : BOOL; //СК открыть
	starter_go : BOOL; //Прокрутка двигателя стартером
	cmd_sh_nIgnition : BOOL; //Взвод защиты по не розжигу на пуске
	cmd_AZ_On : BOOL; //Включение зажигания
	cmd_sh_nBoost : BOOL; //Взвод защиты по не раскрутке
	cmd_VS_Off : BOOL; //Останов воздушного стартера
	cmd_KR11_Off : BOOL; //Закрытие крана 11, открытие крана 10
	cmd_PNU_Off : BOOL; //Отключение маслонасоса уплотнения
	cmd_PNS_Off : BOOL; //Отключение маслонасоса смазки
	cmd_KPV234_Off : BOOL; //Закрыть КПВ 2, 3, 4
	heating_end : BOOL; //Прогрев двигателя окончен
	Ntk_Up : BOOL; //Подъём оборотов
	KPV15_close : BOOL; //Закрытие КПВ 1, 5
	finish : BOOL; //Завершение
	{attribute 'symbol' := 'read'}
	drm : Tdrm; //Интерфейсный функциональный блок
END_VAR
VAR
	start : BOOL; //Запуск последовательности
	break : BOOL; //Принудительный выход из последовательности
END_VAR

                    //Собираем переходы для визуализации
drm.transition.0 := start := APK.cmd_start_D; //Запуск последовательности (0→1): АПК => Пуск двигателя
drm.transition.1 := am.KR11.isOn AND am.KR10.isOff; //1→2: Кран 11 открылся, кран 10 закрылся
drm.transition.2 := acpar.Ntk.value < 100.0; //2→3: Nтк < 100 об/мин
drm.transition.3 := am.KR12.isON AND am.KR9.isOff; //3→4: Продувка топливного газа
drm.transition.4 := aipar.Ptg_inTRK.value > 1.96 AND NOT dipar.Pm_SAR_An.value AND acpar.Ntk.value > 1800; //4→5: Давление ТГ > 20 кгс/см2 И Pm перед ДГ > 15 кгс/см2 И Ntk > 1800 об/мин
drm.transition.5 := acpar.Ntk.value > 4500; //5→6: Nтк > 4500 об/мин
drm.transition.6 := FuelReg.fReg.heating; //6→7: Переход двигателя в режим прогрева
drm.transition.7 := NOT FuelReg.fReg.heating; //7→8: Прогрев двигателя
drm.transition.8 := am.KPV1.isOff AND am.KPV5.isOff; //8→9: Закрытие КПВ
drm.transition.9 := TRUE; //9→0: Логическая 1
drm.transition.31 := break := alg.AO; //Принудительный выход из последовательности (N→0): Режимы аварийного останова

//Вызываем экземпляр интерфейсного функционального блока
drm(cycle := cycle);

CASE drm.step OF
-1:	//Сброс команд с предыдущих шагов
	finish := FALSE;
	//Условие запуска последовательности
	//АПК => Пуск двигателя
	IF start AND NOT break THEN drm.step := 1; END_IF;
1:	//Запись уставки таймера шага
	drm.step := 1;//Текущий шаг
	drm.timer_pt := cycle; //Таймер: один цикл вызова

	//Команды текущего шага
	(*1*) cmd_KR11_On := drm.cmd.0 := TRUE; //Открытие крана 11, закрытие крана 10
	(*1*) drm.error.0 := am.KR11.notOn OR am.KR10.notOff; //Кран 11 не открылся, кран 10 не закрылся

	//Условие перехода (1)→(2)
	//Кран 11 открылся, кран 10 закрылся
	IF (am.KR11.isOn AND am.KR10.isOff) AND drm.timeout THEN
		drm.cmd := drm.error := 0; drm.timer_pt := cycle; drm.inc := FALSE; drm.step := 2;
		cmd_KR11_On := FALSE; //Открытие крана 11, закрытие крана 10
	END_IF;
2:	//Запись уставки таймера шага
	drm.step := 2;//Текущий шаг
	drm.timer_pt := cycle; //Таймер: один цикл вызова

	//Команды текущего шага
	(*1*) check_Ntk := drm.cmd.0 := TRUE; //Проверка Nтк
	(*1*) drm.error.0 := acpar.Ntk.value > 100.0; //Nтк > 100 об/мин

	//Условие перехода (2)→(3)
	//Nтк < 100 об/мин
	IF (acpar.Ntk.value < 100.0) AND drm.timeout THEN
		drm.cmd := drm.error := 0; drm.timer_pt := cycle; drm.inc := FALSE; drm.step := 3;
		check_Ntk := FALSE; //Проверка Nтк
	END_IF;
3:	//Запись уставки таймера шага
	drm.step := 3;//Текущий шаг
	drm.timer_pt := cycle; //Таймер: один цикл вызова

	//Команды текущего шага
	(*1*) cmd_KR12_On := drm.cmd.0 := TRUE; //Открытие крана 12, закрытие крана 9
	(*1*) drm.error.0 := am.KR12.notOn OR am.KR9.notOff; //Кран 12 не открылся, кран 9 не закрылся

	(*2*) cmd_VNA_On := drm.cmd.1 := TRUE; //Включение Э/М ВНА

	(*3*) cmd_KPV_On := drm.cmd.2 := TRUE; //Открыть КПВ

	(*4*) cmd_VS_On := drm.cmd.3 := TRUE; //Пуск воздушного стартера
	(*4*) drm.error.3 := am.KR13.notOn; //Кран 13 не открылся

	//Условие перехода (3)→(4)
	//Продувка топливного газа
	IF (am.KR12.isON AND am.KR9.isOff) AND drm.timeout THEN
		drm.cmd := drm.error := 0; drm.timer_pt := cycle; drm.inc := FALSE; drm.step := 4;
		cmd_KR12_On := FALSE; //Открытие крана 12, закрытие крана 9
		cmd_KPV_On := FALSE; //Открыть КПВ
		cmd_VS_On := FALSE; //Пуск воздушного стартера
	END_IF;
4:	//Запись уставки таймера шага
	drm.step := 4;//Текущий шаг
	drm.timer_pt := cycle; //Таймер: один цикл вызова

	//Команды текущего шага
	(*1*) cmd_sh_TG_On := drm.cmd.0 := TRUE; //Взвести защиту по ТГ

	(*2*) cmd_SK_On := drm.cmd.1 := TRUE; //СК открыть

	(*3*) starter_go := drm.cmd.2 := TRUE; //Прокрутка двигателя стартером

	//Условие перехода (4)→(5)
	//Давление ТГ > 20 кгс/см2 И Pm перед ДГ > 15 кгс/см2 И Ntk > 1800 об/мин
	IF (aipar.Ptg_inTRK.value > 1.96 AND NOT dipar.Pm_SAR_An.value AND acpar.Ntk.value > 1800) AND drm.timeout THEN
		drm.cmd := drm.error := 0; drm.timer_pt := cycle; drm.inc := FALSE; drm.step := 5;
		cmd_sh_TG_On := FALSE; //Взвести защиту по ТГ
		cmd_SK_On := FALSE; //СК открыть
		starter_go := FALSE; //Прокрутка двигателя стартером
	END_IF;
5:	//Запись уставки таймера шага
	drm.step := 5;//Текущий шаг
	drm.timer_pt := cycle; //Таймер: один цикл вызова

	//Команды текущего шага
	(*1*) am.KR15.on := drm.cmd.0 := TRUE; //Открытие крана 15

	(*2*) cmd_sh_nIgnition := drm.cmd.1 := TRUE; //Взвод защиты по не розжигу на пуске

	(*3*) cmd_AZ_On := drm.cmd.2 := drm.step_time <= cycle; //Включение зажигания

	(*4*) FuelReg.fReg.startCom := drm.cmd.3 := TRUE; //Пуск двигателя

	//Условие перехода (5)→(6)
	//Nтк > 4500 об/мин
	IF (acpar.Ntk.value > 4500) AND drm.timeout THEN
		drm.cmd := drm.error := 0; drm.timer_pt := cycle; drm.inc := FALSE; drm.step := 6;
		cmd_sh_nIgnition := FALSE; //Взвод защиты по не розжигу на пуске
		cmd_AZ_On := FALSE; //Включение зажигания
		FuelReg.fReg.startCom := FALSE; //Пуск двигателя
	END_IF;
6:	//Запись уставки таймера шага
	drm.step := 6;//Текущий шаг
	drm.timer_pt := 10; //Таймер: 10 секунд

	//Команды текущего шага
	(*1*) cmd_sh_nBoost := drm.cmd.0 := drm.step_time <= cycle; //Взвод защиты по не раскрутке

	(*2*) cmd_VS_Off := drm.cmd.1 := TRUE; //Останов воздушного стартера
	(*2*) drm.error.1 := am.KR13.notOff; //Кран 13 не закрылся

	(*3*) cmd_KR11_Off := drm.cmd.2 := TRUE; //Закрытие крана 11, открытие крана 10
	(*3*) drm.error.2 := am.KR11.notOff OR am.KR10.notOn; //Кран 11 не закрылся, кран 10 не открылся

	(*4*) am.KR15.on := FALSE; //Кран 15 закрыть

	//Условие перехода (6)→(7)
	//Переход двигателя в режим прогрева
	IF (FuelReg.fReg.heating) AND drm.timeout THEN
		drm.cmd := drm.error := 0; drm.timer_pt := cycle; drm.inc := FALSE; drm.step := 7;
		cmd_sh_nBoost := FALSE; //Взвод защиты по не раскрутке
		cmd_VS_Off := FALSE; //Останов воздушного стартера
		cmd_KR11_Off := FALSE; //Закрытие крана 11, открытие крана 10
	END_IF;
7:	//Запись уставки таймера шага
	drm.step := 7;//Текущий шаг
	drm.inc := TRUE; //Выставляем признак инкремента

	//Команды текущего шага
	(*1*) cmd_VNA_On := FALSE; //Отключение Э/М ВНА

	(*2*) cmd_PNU_Off := drm.cmd.1 := drm.step_time <= cycle; //Отключение маслонасоса уплотнения
	(*2*) drm.error.1 := am.PNU.notOff; //Маслонасос уплотнений не выключился

	(*3*) cmd_PNS_Off := drm.cmd.2 := drm.step_time <= cycle; //Отключение маслонасоса смазки
	(*3*) drm.error.2 := am.PNS.notOff; //Маслонасос смазки не выключился

	(*4*) cmd_KPV234_Off := drm.cmd.3 := drm.step_time <= cycle; //Закрыть КПВ 2, 3, 4
	(*4*) drm.error.3 := am.KPV2.notOff AND am.KPV3.notOff AND am.KPV4.notOff; //КПВ 2, 3, 4 не закрылись

	//Условие перехода (7)→(8)
	//Прогрев двигателя
	IF (NOT FuelReg.fReg.heating) AND drm.timeout THEN
		drm.cmd := drm.error := 0; drm.timer_pt := cycle; drm.inc := FALSE; drm.step := 8;
		cmd_PNU_Off := FALSE; //Отключение маслонасоса уплотнения
		cmd_PNS_Off := FALSE; //Отключение маслонасоса смазки
		cmd_KPV234_Off := FALSE; //Закрыть КПВ 2, 3, 4
	END_IF;
8:	//Запись уставки таймера шага
	drm.step := 8;//Текущий шаг
	drm.timer_pt := cycle; //Таймер: один цикл вызова

	//Команды текущего шага
	(*1*) cmd_AZ_On := drm.cmd.0 := drm.step_time <= cycle; //Тренирование свечей зажигания

	(*2*) heating_end := drm.cmd.1 := TRUE; //Прогрев двигателя окончен

	(*3*) Ntk_Up := drm.cmd.2 := TRUE; //Подъём оборотов

	(*4*) KPV15_close := drm.cmd.3 := TRUE; //Закрытие КПВ 1, 5
	(*4*) drm.error.3 := am.KPV1.notOff AND am.KPV5.notOff; //КПВ 1, 5 не закрылись

	//Условие перехода (8)→(9)
	//Закрытие КПВ
	IF (am.KPV1.isOff AND am.KPV5.isOff) AND drm.timeout THEN
		drm.cmd := drm.error := 0; drm.timer_pt := cycle; drm.inc := FALSE; drm.step := 9;
		cmd_AZ_On := FALSE; //Тренирование свечей зажигания
		heating_end := FALSE; //Прогрев двигателя окончен
		Ntk_Up := FALSE; //Подъём оборотов
		KPV15_close := FALSE; //Закрытие КПВ 1, 5
	END_IF;
9:	//Запись уставки таймера шага
	drm.step := 9;//Текущий шаг
	drm.timer_pt := cycle; //Таймер: один цикл вызова

	//Команды текущего шага
	(*1*) finish := drm.cmd.0 := TRUE; //Завершение

	//Условие перехода (9)→(0)
	//Логическая 1
	IF (TRUE) AND drm.timeout THEN
		drm.cmd := drm.error := 0; drm.timer_pt := cycle; drm.inc := FALSE; drm.step := -1;
		finish := FALSE; //Завершение
	END_IF;
END_CASE

//Принудительный выход из последовательности
IF break THEN
	drm.step := -1; drm.cmd := drm.error := 0; drm.timer_pt := cycle; drm.inc := FALSE;
	cmd_KR11_On := FALSE; //Открытие крана 11, закрытие крана 10
	check_Ntk := FALSE; //Проверка Nтк
	cmd_KR12_On := FALSE; //Открытие крана 12, закрытие крана 9
	cmd_VNA_On := FALSE; //Включение Э/М ВНА
	cmd_KPV_On := FALSE; //Открыть КПВ
	cmd_VS_On := FALSE; //Пуск воздушного стартера
	cmd_sh_TG_On := FALSE; //Взвести защиту по ТГ
	cmd_SK_On := FALSE; //СК открыть
	starter_go := FALSE; //Прокрутка двигателя стартером
	am.KR15.on := FALSE; //Открытие крана 15
	cmd_sh_nIgnition := FALSE; //Взвод защиты по не розжигу на пуске
	cmd_AZ_On := FALSE; //Включение зажигания
	FuelReg.fReg.startCom := FALSE; //Пуск двигателя
	cmd_sh_nBoost := FALSE; //Взвод защиты по не раскрутке
	cmd_VS_Off := FALSE; //Останов воздушного стартера
	cmd_KR11_Off := FALSE; //Закрытие крана 11, открытие крана 10
	cmd_PNU_Off := FALSE; //Отключение маслонасоса уплотнения
	cmd_PNS_Off := FALSE; //Отключение маслонасоса смазки
	cmd_KPV234_Off := FALSE; //Закрыть КПВ 2, 3, 4
	cmd_AZ_On := FALSE; //Тренирование свечей зажигания
	heating_end := FALSE; //Прогрев двигателя окончен
	Ntk_Up := FALSE; //Подъём оборотов
	KPV15_close := FALSE; //Закрытие КПВ 1, 5
	finish := FALSE; //Завершение
END_IF;

                  
END_FUNCTION_BLOCK

{region INFO}
(*
 Назначение: вызов функциональных блоков последовательностей подсистемы "Газовая обвязка"
 Автор: /Разработчик/ 08.08.2025 9:04:03
 Версия: v00.00.18
 Проект: KA107
*)
{endregion}
FUNCTION go_update : BOOL
VAR_INPUT
	cycle : REAL; //цикл вызова
END_VAR

                    //Заполнение контура компрессора
Filling(cycle := cycle);
 //Стравливание контура компрессора
Bleeding(cycle := cycle);

                  
END_FUNCTION

{region INFO}
(*
 Наименование последовательности: Стравливание контура компрессора
 Автор: /Разработчик/ 08.08.2025 9:04:03
 Версия: v00.00.18
 Проект: KA107
*)
{endregion}
{attribute 'symbol' := 'none'}
FUNCTION_BLOCK PUBLIC T_Bleeding
VAR_INPUT
	cycle : REAL; //цикл вызова
END_VAR
VAR_OUTPUT
	cmd_Kr4_Off : BOOL; //Кран 4 закрыть
	cmd_Kr1_Off : BOOL; //Кран 1 закрыть
	cmd_Kr2_Off : BOOL; //Кран 2 закрыть
	cmd_Kr6_Off : BOOL; //Кран 6 закрыть
	cmd_Kr5_On : BOOL; //Кран 5 открыть
	bleeding : BOOL; //Стравливание
	finish : BOOL; //Завершение
	{attribute 'symbol' := 'read'}
	drm : Tdrm; //Интерфейсный функциональный блок
END_VAR
VAR
	start : BOOL; //Запуск последовательности
	break : BOOL; //Принудительный выход из последовательности
END_VAR

                    //Собираем переходы для визуализации
drm.transition.0 := start := AOss.cmd_bleeding OR NOss.cmd_bleeding OR Bleeding_full.cmd_bleeding; //Запуск последовательности (0→1): (АОсс => Стравливание) ИЛИ (НОсс => Стравливание) ИЛИ (Стравливание => Стравливание)
drm.transition.1 := am.Kr4.isOFF AND am.Kr1.isOFF AND am.Kr2.isOFF AND am.Kr6.isOFF; //1→2: Кран 4 закрыт И Кран 1 закрыт И Кран 2 закрыт И Кран 6 закрыт
drm.transition.2 := am.Kr5.isON AND aipar.Pg_inN.value < 0.2; //2→3: Кран 5 открыт И Р газа на входе К < 0.2 МПа
drm.transition.3 := TRUE; //3→0: Логическая 1
drm.transition.31 := break := NOT mde.NOss AND NOT mde.AOss AND NOT bleeding_full.drm.active; //Принудительный выход из последовательности (N→0): Отсутствие запускающих режимов

//Вызываем экземпляр интерфейсного функционального блока
drm(cycle := cycle);

CASE drm.step OF
-1:	//Сброс команд с предыдущих шагов
	finish := FALSE;
	//Условие запуска последовательности
	//(АОсс => Стравливание) ИЛИ (НОсс => Стравливание) ИЛИ (Стравливание => Стравливание)
	IF start AND NOT break THEN drm.step := 1; END_IF;
1:	//Запись уставки таймера шага
	drm.step := 1;//Текущий шаг
	drm.timer_pt := cycle; //Таймер: один цикл вызова

	//Команды текущего шага
	(*1*) cmd_Kr4_Off := drm.cmd.0 := TRUE; //Кран 4 закрыть
	(*1*) drm.error.0 := am.Kr4.notOff; //Кран 4 не закрылся

	(*2*) cmd_Kr1_Off := drm.cmd.1 := TRUE; //Кран 1 закрыть
	(*2*) drm.error.1 := am.Kr1.notOff; //Кран 1 не закрылся

	(*3*) cmd_Kr2_Off := drm.cmd.2 := TRUE; //Кран 2 закрыть
	(*3*) drm.error.2 := am.Kr2.notOff; //Кран 2 не закрылся

	(*4*) cmd_Kr6_Off := drm.cmd.3 := TRUE; //Кран 6 закрыть
	(*4*) drm.error.3 := am.Kr6.notOff; //Кран 6 не закрылся

	//Условие перехода (1)→(2)
	//Кран 4 закрыт И Кран 1 закрыт И Кран 2 закрыт И Кран 6 закрыт
	IF (am.Kr4.isOFF AND am.Kr1.isOFF AND am.Kr2.isOFF AND am.Kr6.isOFF) AND drm.timeout THEN
		drm.cmd := drm.error := 0; drm.timer_pt := cycle; drm.inc := FALSE; drm.step := 2;
		cmd_Kr4_Off := FALSE; //Кран 4 закрыть
		cmd_Kr1_Off := FALSE; //Кран 1 закрыть
		cmd_Kr2_Off := FALSE; //Кран 2 закрыть
		cmd_Kr6_Off := FALSE; //Кран 6 закрыть
	END_IF;
2:	//Запись уставки таймера шага
	drm.step := 2;//Текущий шаг
	drm.timer_pt := cycle; //Таймер: один цикл вызова

	//Команды текущего шага
	(*1*) cmd_Kr5_On := drm.cmd.0 := TRUE; //Кран 5 открыть
	(*1*) drm.error.0 := am.Kr5.notOn; //Кран 5 не открылся

	(*2*) bleeding := drm.cmd.1 := TRUE; //Стравливание
	(*2*) drm.error.1 := aipar.Pg_inN.value > 0.2; //Р газа на входе К > 0.2 МПа

	//Условие перехода (2)→(3)
	//Кран 5 открыт И Р газа на входе К < 0.2 МПа
	IF (am.Kr5.isON AND aipar.Pg_inN.value < 0.2) AND drm.timeout THEN
		drm.cmd := drm.error := 0; drm.timer_pt := cycle; drm.inc := FALSE; drm.step := 3;
		cmd_Kr5_On := FALSE; //Кран 5 открыть
		bleeding := FALSE; //Стравливание
	END_IF;
3:	//Запись уставки таймера шага
	drm.step := 3;//Текущий шаг
	drm.timer_pt := cycle; //Таймер: один цикл вызова

	//Команды текущего шага
	(*1*) finish := drm.cmd.0 := TRUE; //Завершение

	//Условие перехода (3)→(0)
	//Логическая 1
	IF (TRUE) AND drm.timeout THEN
		drm.cmd := drm.error := 0; drm.timer_pt := cycle; drm.inc := FALSE; drm.step := -1;
		finish := FALSE; //Завершение
	END_IF;
END_CASE

//Принудительный выход из последовательности
IF break THEN
	drm.step := -1; drm.cmd := drm.error := 0; drm.timer_pt := cycle; drm.inc := FALSE;
	cmd_Kr4_Off := FALSE; //Кран 4 закрыть
	cmd_Kr1_Off := FALSE; //Кран 1 закрыть
	cmd_Kr2_Off := FALSE; //Кран 2 закрыть
	cmd_Kr6_Off := FALSE; //Кран 6 закрыть
	cmd_Kr5_On := FALSE; //Кран 5 открыть
	bleeding := FALSE; //Стравливание
	finish := FALSE; //Завершение
END_IF;

                  
END_FUNCTION_BLOCK

{region INFO}
(*
 Наименование последовательности: Заполнение контура компрессора
 Автор: /Разработчик/ 08.08.2025 9:04:03
 Версия: v00.00.18
 Проект: KA107
*)
{endregion}
{attribute 'symbol' := 'none'}
FUNCTION_BLOCK PUBLIC T_Filling
VAR_INPUT
	cycle : REAL; //цикл вызова
END_VAR
VAR_OUTPUT
	cmd_Kr4_On : BOOL; //Кран 4 открыть
	purge : BOOL; //Продувка контура нагнетателя
	cmd_Kr5_Off : BOOL; //Кран 5 закрыть
	filling : BOOL; //Заполнение
	Pg_Ok : BOOL; //Давление в контуре 30 кгс/см2
	stab : BOOL; //Стабилизация
	cmd_Kr1_On : BOOL; //Кран 1 открыть
	cmd_Kr6_On : BOOL; //Кран 6 открыть
	cmd_Kr4_Off : BOOL; //Кран 4 закрыть
	finish : BOOL; //Завершение
	{attribute 'symbol' := 'read'}
	drm : Tdrm; //Интерфейсный функциональный блок
END_VAR
VAR
	start : BOOL; //Запуск последовательности
	break : BOOL; //Принудительный выход из последовательности
END_VAR

                    //Собираем переходы для визуализации
drm.transition.0 := start := KPK.cmd_filling OR APK.cmd_filling; //Запуск последовательности (0→1): (КПК => Заполнение) ИЛИ (АПК => Заполнение)
drm.transition.1 := am.Kr4.isON; //1→2: Кран 4 открыт
drm.transition.2 := TRUE; //2→3: Логическая 1
drm.transition.3 := am.Kr5.isOFF; //3→4: Кран 5 закрыт
drm.transition.4 := alg.nIncPgN AND aipar.Pg_outN.value > 2.942; //4→5: Рост давления в контуре > 0.2 МПа в секунду И давление в контуре > 30 кгс/см2
drm.transition.5 := TRUE; //5→6: Логическая 1
drm.transition.6 := am.Kr1.isON; //6→7: Кран 1 открыт
drm.transition.7 := am.Kr4.isOFF; //7→8: Кран 4 закрыт
drm.transition.8 := TRUE; //8→0: Логическая 1
drm.transition.31 := break := alg.AO; //Принудительный выход из последовательности (N→0): Режимы аварийного останова

//Вызываем экземпляр интерфейсного функционального блока
drm(cycle := cycle);

CASE drm.step OF
-1:	//Сброс команд с предыдущих шагов
	finish := FALSE;
	//Условие запуска последовательности
	//(КПК => Заполнение) ИЛИ (АПК => Заполнение)
	IF start AND NOT break THEN drm.step := 1; END_IF;
1:	//Запись уставки таймера шага
	drm.step := 1;//Текущий шаг
	drm.timer_pt := cycle; //Таймер: один цикл вызова

	//Команды текущего шага
	(*1*) cmd_Kr4_On := drm.cmd.0 := TRUE; //Кран 4 открыть
	(*1*) drm.error.0 := am.Kr4.notOn; //Кран 4 не открылся

	//Условие перехода (1)→(2)
	//Кран 4 открыт
	IF (am.Kr4.isON) AND drm.timeout THEN
		drm.cmd := drm.error := 0; drm.timer_pt := cycle; drm.inc := FALSE; drm.step := 2;
		cmd_Kr4_On := FALSE; //Кран 4 открыть
	END_IF;
2:	//Запись уставки таймера шага
	drm.step := 2;//Текущий шаг
	drm.timer_pt := 10; //Таймер: 10 секунд

	//Команды текущего шага
	(*1*) purge := drm.cmd.0 := TRUE; //Продувка контура нагнетателя

	//Условие перехода (2)→(3)
	//Логическая 1
	IF (TRUE) AND drm.timeout THEN
		drm.cmd := drm.error := 0; drm.timer_pt := cycle; drm.inc := FALSE; drm.step := 3;
		purge := FALSE; //Продувка контура нагнетателя
	END_IF;
3:	//Запись уставки таймера шага
	drm.step := 3;//Текущий шаг
	drm.timer_pt := cycle; //Таймер: один цикл вызова

	//Команды текущего шага
	(*1*) cmd_Kr5_Off := drm.cmd.0 := TRUE; //Кран 5 закрыть
	(*1*) drm.error.0 := am.Kr5.notOff; //Кран 5 не закрылся

	//Условие перехода (3)→(4)
	//Кран 5 закрыт
	IF (am.Kr5.isOFF) AND drm.timeout THEN
		drm.cmd := drm.error := 0; drm.timer_pt := cycle; drm.inc := FALSE; drm.step := 4;
		cmd_Kr5_Off := FALSE; //Кран 5 закрыть
	END_IF;
4:	//Запись уставки таймера шага
	drm.step := 4;//Текущий шаг
	drm.timer_pt := cycle; //Таймер: один цикл вызова

	//Команды текущего шага
	(*1*) filling := drm.cmd.0 := TRUE; //Заполнение
	(*1*) drm.error.0 := NOT  alg.nIncPgN; //Прирост давления в контуре > 0.05 МПа в секунду 

	(*2*) Pg_Ok := drm.cmd.1 := TRUE; //Давление в контуре 30 кгс/см2
	(*2*) drm.error.1 := aipar.Pg_outN.value < 2.942; //Давление в контуре < 30 кгс/см2

	//Условие перехода (4)→(5)
	//Рост давления в контуре > 0.2 МПа в секунду И давление в контуре > 30 кгс/см2
	IF (alg.nIncPgN AND aipar.Pg_outN.value > 2.942) AND drm.timeout THEN
		drm.cmd := drm.error := 0; drm.timer_pt := cycle; drm.inc := FALSE; drm.step := 5;
		filling := FALSE; //Заполнение
		Pg_Ok := FALSE; //Давление в контуре 30 кгс/см2
	END_IF;
5:	//Запись уставки таймера шага
	drm.step := 5;//Текущий шаг
	drm.timer_pt := 20; //Таймер: 20 секунд

	//Команды текущего шага
	(*1*) stab := drm.cmd.0 := TRUE; //Стабилизация

	//Условие перехода (5)→(6)
	//Логическая 1
	IF (TRUE) AND drm.timeout THEN
		drm.cmd := drm.error := 0; drm.timer_pt := cycle; drm.inc := FALSE; drm.step := 6;
		stab := FALSE; //Стабилизация
	END_IF;
6:	//Запись уставки таймера шага
	drm.step := 6;//Текущий шаг
	drm.timer_pt := cycle; //Таймер: один цикл вызова

	//Команды текущего шага
	(*1*) cmd_Kr1_On := drm.cmd.0 := TRUE; //Кран 1 открыть
	(*1*) drm.error.0 := am.Kr1.notOn; //Кран 1 не открылся

	(*2*) cmd_Kr6_On := drm.cmd.1 := TRUE; //Кран 6 открыть
	(*2*) drm.error.1 := am.Kr6.notOn; //Кран 6 не открылся

	//Условие перехода (6)→(7)
	//Кран 1 открыт
	IF (am.Kr1.isON) AND drm.timeout THEN
		drm.cmd := drm.error := 0; drm.timer_pt := cycle; drm.inc := FALSE; drm.step := 7;
		cmd_Kr1_On := FALSE; //Кран 1 открыть
		cmd_Kr6_On := FALSE; //Кран 6 открыть
	END_IF;
7:	//Запись уставки таймера шага
	drm.step := 7;//Текущий шаг
	drm.timer_pt := cycle; //Таймер: один цикл вызова

	//Команды текущего шага
	(*1*) cmd_Kr4_Off := drm.cmd.0 := TRUE; //Кран 4 закрыть
	(*1*) drm.error.0 := am.Kr4.notOff; //Кран 4 не закрылся

	//Условие перехода (7)→(8)
	//Кран 4 закрыт
	IF (am.Kr4.isOFF) AND drm.timeout THEN
		drm.cmd := drm.error := 0; drm.timer_pt := cycle; drm.inc := FALSE; drm.step := 8;
		cmd_Kr4_Off := FALSE; //Кран 4 закрыть
	END_IF;
8:	//Запись уставки таймера шага
	drm.step := 8;//Текущий шаг
	drm.timer_pt := cycle; //Таймер: один цикл вызова

	//Команды текущего шага
	(*1*) finish := drm.cmd.0 := TRUE; //Завершение

	//Условие перехода (8)→(0)
	//Логическая 1
	IF (TRUE) AND drm.timeout THEN
		drm.cmd := drm.error := 0; drm.timer_pt := cycle; drm.inc := FALSE; drm.step := -1;
		finish := FALSE; //Завершение
	END_IF;
END_CASE

//Принудительный выход из последовательности
IF break THEN
	drm.step := -1; drm.cmd := drm.error := 0; drm.timer_pt := cycle; drm.inc := FALSE;
	cmd_Kr4_On := FALSE; //Кран 4 открыть
	purge := FALSE; //Продувка контура нагнетателя
	cmd_Kr5_Off := FALSE; //Кран 5 закрыть
	filling := FALSE; //Заполнение
	Pg_Ok := FALSE; //Давление в контуре 30 кгс/см2
	stab := FALSE; //Стабилизация
	cmd_Kr1_On := FALSE; //Кран 1 открыть
	cmd_Kr6_On := FALSE; //Кран 6 открыть
	cmd_Kr4_Off := FALSE; //Кран 4 закрыть
	finish := FALSE; //Завершение
END_IF;

                  
END_FUNCTION_BLOCK

{region INFO}
(*
 Назначение: вызов функциональных блоков последовательностей подрежимов
 Автор: /Разработчик/ 08.08.2025 9:04:03
 Версия: v00.00.18
 Проект: KA107
*)
{endregion}
FUNCTION smd_update : BOOL
VAR_INPUT
	cycle : REAL; //цикл вызова
END_VAR

                    //ХП
HP(cycle := cycle);

 //КПК
KPK(cycle := cycle);

 //АПК
APK(cycle := cycle);

 //Переход К-М
K_M(cycle := cycle);

 //Переход М-К
M_K(cycle := cycle);

 //НОсс
NOss(cycle := cycle);

 //НОбс
NObs(cycle := cycle);

 //АОсс
AOss(cycle := cycle);

 //АОбс
AObs(cycle := cycle);

 //Стравливание
Bleeding_full(cycle := cycle);

 //Контроль САУ
Check_SAU(cycle := cycle);

 //Комплексное тестирование
testing(cycle := cycle);

                  
END_FUNCTION

{region INFO}
(*
 Наименование последовательности: АОбс
 Автор: /Разработчик/ 08.08.2025 9:04:03
 Версия: v00.00.18
 Проект: KA107
*)
{endregion}
{attribute 'symbol' := 'none'}
FUNCTION_BLOCK PUBLIC T_AObs
VAR_INPUT
	cycle : REAL; //цикл вызова
END_VAR
VAR_OUTPUT
	emergStopCom : BOOL; //Аварийный останов двигателя
	cmd_M_K : BOOL; //Запуск последовательности "Переход М-К"
	sh_ms_off : BOOL; //Снятие защиты по маслосистеме ТК и СТ
	cmd_KPV15_On : BOOL; //Открыть КПВ 1, 5
	cmd_KPV234_On : BOOL; //Открыть КПВ 2, 3, 4
	cmd_VNA_On : BOOL; //Включение Э/М ВНА
	cmd_sh_TG_Off : BOOL; //Снятие защиты по ТГ
	cmd_PNU_S_On : BOOL; //Включение маслонасосов смазки и уплотнения
	cmd_KR12_Off : BOOL; //Закрытие крана 12, открытие крана 9
	cmd_VS_Off : BOOL; //Останов воздушного стартера
	cmd_Kr4_Off : BOOL; //Кран 4 закрыть
	cmd_KR11_Off : BOOL; //Закрытие крана 11, открытие крана 10
	check_Nst : BOOL; //Проверка Nст
	check_Ntk : BOOL; //Выбег двигателя
	cmd_Kr1_Off : BOOL; //Кран 1 закрыть
	cmd_Kr2_Off : BOOL; //Кран 2 закрыть
	cmd_Kr6_Off : BOOL; //Кран 6 закрыть
	cmd_Kr4_On : BOOL; //Кран 4 открыть
	finish : BOOL; //Завершение
	{attribute 'symbol' := 'read'}
	drm : Tdrm; //Интерфейсный функциональный блок
END_VAR
VAR
	start : BOOL; //Запуск последовательности
	break : BOOL; //Принудительный выход из последовательности
END_VAR

                    //Собираем переходы для визуализации
drm.transition.0 := start := mde.AObs; //Запуск последовательности (0→1): Режим АОбс
drm.transition.1 := am.Kr4.isOFF AND ( acpar.Nst.value < 100.0 OR acpar.Nst.flt ); //1→2: Кран 4 закрыт И Nст < 100 об/мин
drm.transition.2 := TRUE; //2→3: Логическая 1
drm.transition.3 := am.Kr1.isOFF AND am.Kr2.isOFF AND am.Kr6.isOFF AND am.Kr4.isON; //3→4: Кран 1 закрыт И Кран 2 закрыт И Кран 6 закрыт И Кран 4 открыт
drm.transition.4 := tch.Unlock.value; //4→0: Деблокировка
drm.transition.31 := break := NOT mde.AObs; //Принудительный выход из последовательности (N→0): Снятие режима

//Вызываем экземпляр интерфейсного функционального блока
drm(cycle := cycle);

CASE drm.step OF
-1:	//Сброс команд с предыдущих шагов
	finish := FALSE;
	//Условие запуска последовательности
	//Режим АОбс
	IF start AND NOT break THEN drm.step := 1; END_IF;
1:	//Запись уставки таймера шага
	drm.step := 1;//Текущий шаг
	drm.timer_pt := 10; //Таймер: 10 секунд

	//Команды текущего шага
	(*1*) emergStopCom := drm.cmd.0 := TRUE; //Аварийный останов двигателя

	(*2*) cmd_M_K := drm.cmd.1 := drm.step_time <= cycle; //Запуск последовательности "Переход М-К"

	(*3*) sh_ms_off := drm.cmd.2 := TRUE; //Снятие защиты по маслосистеме ТК и СТ

	(*4*) cmd_KPV15_On := drm.cmd.3 := TRUE; //Открыть КПВ 1, 5
	(*4*) drm.error.3 := am.KPV1.notOn AND am.KPV5.notOn; //КПВ 1, 5 не открылись

	(*5*) cmd_KPV234_On := drm.cmd.4 := TRUE; //Открыть КПВ 2, 3, 4
	(*5*) drm.error.4 := am.KPV2.notOn OR am.KPV3.notOn OR am.KPV4.notOn; //КПВ 2, 3, 4 не открылись

	(*6*) cmd_VNA_On := drm.cmd.5 := TRUE; //Включение Э/М ВНА

	(*7*) cmd_sh_TG_Off := drm.cmd.6 := TRUE; //Снятие защиты по ТГ

	(*8*) cmd_PNU_S_On := drm.cmd.7 := TRUE; //Включение маслонасосов смазки и уплотнения

	(*9*) cmd_KR12_Off := drm.cmd.8 := TRUE; //Закрытие крана 12, открытие крана 9
	(*9*) drm.error.8 := am.KR12.notOff OR am.KR9.notOn; //Кран 12 не закрылся, кран 9 не открылся

	(*10*) cmd_VS_Off := drm.cmd.9 := TRUE; //Останов воздушного стартера
	(*10*) drm.error.9 := am.KR13.notOff; //Кран 13 не закрылся

	(*11*) am.KR15.on := FALSE; //Кран 15 закрыть
	(*11*) drm.error.10 := am.KR15.notOff; //Кран 15 не закрылся

	(*12*) cmd_Kr4_Off := drm.cmd.11 := TRUE; //Кран 4 закрыть
	(*12*) drm.error.11 := am.Kr4.notOff; //Кран 4 не закрылся

	(*13*) cmd_KR11_Off := drm.cmd.12 := TRUE; //Закрытие крана 11, открытие крана 10

	(*14*) check_Nst := drm.cmd.13 := TRUE; //Проверка Nст
	(*14*) drm.error.13 := acpar.Nst.value > 100.0; //Nст > 100 об/мин

	//Условие перехода (1)→(2)
	//Кран 4 закрыт И Nст < 100 об/мин
	IF (am.Kr4.isOFF AND ( acpar.Nst.value < 100.0 OR acpar.Nst.flt )) AND drm.timeout THEN
		drm.cmd := drm.error := 0; drm.timer_pt := cycle; drm.inc := FALSE; drm.step := 2;
		cmd_M_K := FALSE; //Запуск последовательности "Переход М-К"
		sh_ms_off := FALSE; //Снятие защиты по маслосистеме ТК и СТ
		cmd_KPV15_On := FALSE; //Открыть КПВ 1, 5
		cmd_KPV234_On := FALSE; //Открыть КПВ 2, 3, 4
		cmd_sh_TG_Off := FALSE; //Снятие защиты по ТГ
		cmd_PNU_S_On := FALSE; //Включение маслонасосов смазки и уплотнения
		cmd_KR12_Off := FALSE; //Закрытие крана 12, открытие крана 9
		cmd_VS_Off := FALSE; //Останов воздушного стартера
		cmd_Kr4_Off := FALSE; //Кран 4 закрыть
		cmd_KR11_Off := FALSE; //Закрытие крана 11, открытие крана 10
		check_Nst := FALSE; //Проверка Nст
	END_IF;
2:	//Запись уставки таймера шага
	drm.step := 2;//Текущий шаг
	drm.timer_pt := 60; //Таймер: 60 секунд

	//Команды текущего шага
	(*1*) check_Ntk := drm.cmd.0 := TRUE; //Выбег двигателя

	//Условие перехода (2)→(3)
	//Логическая 1
	IF (TRUE) AND drm.timeout THEN
		drm.cmd := drm.error := 0; drm.timer_pt := cycle; drm.inc := FALSE; drm.step := 3;
		check_Ntk := FALSE; //Выбег двигателя
	END_IF;
3:	//Запись уставки таймера шага
	drm.step := 3;//Текущий шаг
	drm.timer_pt := cycle; //Таймер: один цикл вызова

	//Команды текущего шага
	(*1*) cmd_VNA_On := FALSE; //Отключение Э/М ВНА

	(*2*) cmd_Kr1_Off := drm.cmd.1 := TRUE; //Кран 1 закрыть
	(*2*) drm.error.1 := am.Kr1.notOff; //Кран 1 не закрылся

	(*3*) cmd_Kr2_Off := drm.cmd.2 := TRUE; //Кран 2 закрыть
	(*3*) drm.error.2 := am.Kr2.notOff; //Кран 2 не закрылся

	(*4*) cmd_Kr6_Off := drm.cmd.3 := TRUE; //Кран 6 закрыть
	(*4*) drm.error.3 := am.Kr6.notOff; //Кран 6 не закрылся

	(*5*) cmd_Kr4_On := drm.cmd.4 := TRUE; //Кран 4 открыть
	(*5*) drm.error.4 := am.Kr4.notOn; //Кран 4 не открылся

	//Условие перехода (3)→(4)
	//Кран 1 закрыт И Кран 2 закрыт И Кран 6 закрыт И Кран 4 открыт
	IF (am.Kr1.isOFF AND am.Kr2.isOFF AND am.Kr6.isOFF AND am.Kr4.isON) AND drm.timeout THEN
		drm.cmd := drm.error := 0; drm.timer_pt := cycle; drm.inc := FALSE; drm.step := 4;
		cmd_Kr1_Off := FALSE; //Кран 1 закрыть
		cmd_Kr2_Off := FALSE; //Кран 2 закрыть
		cmd_Kr6_Off := FALSE; //Кран 6 закрыть
		cmd_Kr4_On := FALSE; //Кран 4 открыть
	END_IF;
4:	//Запись уставки таймера шага
	drm.step := 4;//Текущий шаг
	drm.timer_pt := cycle; //Таймер: один цикл вызова

	//Команды текущего шага
	(*1*) finish := drm.cmd.0 := TRUE; //Завершение
	(*1*) drm.error.0 := NOT tch.Unlock.value; //АОбс завершен, нажмите кнопку "Деблокировка"

	//Условие перехода (4)→(0)
	//Деблокировка
	IF (tch.Unlock.value) AND drm.timeout THEN
		drm.cmd := drm.error := 0; drm.timer_pt := cycle; drm.inc := FALSE; drm.step := -1;
		finish := FALSE; //Завершение
	END_IF;
END_CASE

//Принудительный выход из последовательности
IF break THEN
	drm.step := -1; drm.cmd := drm.error := 0; drm.timer_pt := cycle; drm.inc := FALSE;
	emergStopCom := FALSE; //Аварийный останов двигателя
	cmd_M_K := FALSE; //Запуск последовательности "Переход М-К"
	sh_ms_off := FALSE; //Снятие защиты по маслосистеме ТК и СТ
	cmd_KPV15_On := FALSE; //Открыть КПВ 1, 5
	cmd_KPV234_On := FALSE; //Открыть КПВ 2, 3, 4
	cmd_VNA_On := FALSE; //Включение Э/М ВНА
	cmd_sh_TG_Off := FALSE; //Снятие защиты по ТГ
	cmd_PNU_S_On := FALSE; //Включение маслонасосов смазки и уплотнения
	cmd_KR12_Off := FALSE; //Закрытие крана 12, открытие крана 9
	cmd_VS_Off := FALSE; //Останов воздушного стартера
	cmd_Kr4_Off := FALSE; //Кран 4 закрыть
	cmd_KR11_Off := FALSE; //Закрытие крана 11, открытие крана 10
	check_Nst := FALSE; //Проверка Nст
	check_Ntk := FALSE; //Выбег двигателя
	cmd_Kr1_Off := FALSE; //Кран 1 закрыть
	cmd_Kr2_Off := FALSE; //Кран 2 закрыть
	cmd_Kr6_Off := FALSE; //Кран 6 закрыть
	cmd_Kr4_On := FALSE; //Кран 4 открыть
	finish := FALSE; //Завершение
END_IF;

                  
END_FUNCTION_BLOCK

{region INFO}
(*
 Наименование последовательности: АОсс
 Автор: /Разработчик/ 08.08.2025 9:04:03
 Версия: v00.00.18
 Проект: KA107
*)
{endregion}
{attribute 'symbol' := 'none'}
FUNCTION_BLOCK PUBLIC T_AOss
VAR_INPUT
	cycle : REAL; //цикл вызова
END_VAR
VAR_OUTPUT
	emergStopCom : BOOL; //Аварийный останов двигателя
	cmd_M_K : BOOL; //Запуск последовательности "Переход М-К"
	sh_ms_off : BOOL; //Снятие защиты по маслосистеме ТК и СТ
	cmd_KPV15_On : BOOL; //Открыть КПВ 1, 5
	cmd_KPV234_On : BOOL; //Открыть КПВ 2, 3, 4
	cmd_VNA_On : BOOL; //Включение Э/М ВНА
	cmd_sh_TG_Off : BOOL; //Снятие защиты по ТГ
	cmd_PNU_S_On : BOOL; //Включение маслонасосов смазки и уплотнения
	cmd_KR12_Off : BOOL; //Закрытие крана 12, открытие крана 9
	cmd_VS_Off : BOOL; //Останов воздушного стартера
	cmd_Kr4_Off : BOOL; //Кран 4 закрыть
	cmd_KR11_Off : BOOL; //Закрытие крана 11, открытие крана 10
	check_Nst : BOOL; //Проверка Nст
	cmd_bleeding : BOOL; //Запуск последовательности "Стравливание контура компрессора"
	check_Ntk : BOOL; //Выбег двигателя
	cmd_shPmN_Off : BOOL; //Снятие защиты по маслосистеме нагнетателя
	cmd_sh_dPmg_Off : BOOL; //Снятие защиты по перепаду "масло-газ"
	cmd_PNU_S_Off : BOOL; //Пуск таймера отключения ПНС, ПНУ
	finish : BOOL; //Завершение
	{attribute 'symbol' := 'read'}
	drm : Tdrm; //Интерфейсный функциональный блок
END_VAR
VAR
	start : BOOL; //Запуск последовательности
	break : BOOL; //Принудительный выход из последовательности
END_VAR

                    //Собираем переходы для визуализации
drm.transition.0 := start := mde.AOss; //Запуск последовательности (0→1): Режим АОсс
drm.transition.1 := am.Kr4.isOFF AND ( acpar.Nst.value < 100.0 OR acpar.Nst.flt ); //1→2: Кран 4 закрыт И Nст < 100 об/мин
drm.transition.2 := bleeding.finish; //2→3: Подрежим "Стравливание контура компрессора" завершен
drm.transition.3 := TRUE; //3→4: Логическая 1
drm.transition.4 := TRUE; //4→5: Логическая 1
drm.transition.5 := TRUE; //5→6: Логическая 1
drm.transition.6 := tch.Unlock.value; //6→0: Деблокировка
drm.transition.31 := break := NOT mde.AOss; //Принудительный выход из последовательности (N→0): Снятие режима

//Вызываем экземпляр интерфейсного функционального блока
drm(cycle := cycle);

CASE drm.step OF
-1:	//Сброс команд с предыдущих шагов
	finish := FALSE;
	//Условие запуска последовательности
	//Режим АОсс
	IF start AND NOT break THEN drm.step := 1; END_IF;
1:	//Запись уставки таймера шага
	drm.step := 1;//Текущий шаг
	drm.timer_pt := 10; //Таймер: 10 секунд

	//Команды текущего шага
	(*1*) emergStopCom := drm.cmd.0 := TRUE; //Аварийный останов двигателя

	(*2*) cmd_M_K := drm.cmd.1 := drm.step_time <= cycle; //Запуск последовательности "Переход М-К"

	(*3*) sh_ms_off := drm.cmd.2 := TRUE; //Снятие защиты по маслосистеме ТК и СТ

	(*4*) cmd_KPV15_On := drm.cmd.3 := TRUE; //Открыть КПВ 1, 5
	(*4*) drm.error.3 := am.KPV1.notOn AND am.KPV5.notOn; //КПВ 1, 5 не открылись

	(*5*) cmd_KPV234_On := drm.cmd.4 := TRUE; //Открыть КПВ 2, 3, 4
	(*5*) drm.error.4 := am.KPV2.notOn OR am.KPV3.notOn OR am.KPV4.notOn; //КПВ 2, 3, 4 не открылись

	(*6*) cmd_VNA_On := drm.cmd.5 := TRUE; //Включение Э/М ВНА

	(*7*) cmd_sh_TG_Off := drm.cmd.6 := TRUE; //Снятие защиты по ТГ

	(*8*) cmd_PNU_S_On := drm.cmd.7 := TRUE; //Включение маслонасосов смазки и уплотнения

	(*9*) cmd_KR12_Off := drm.cmd.8 := TRUE; //Закрытие крана 12, открытие крана 9
	(*9*) drm.error.8 := am.KR12.notOff OR am.KR9.notOn; //Кран 12 не закрылся, кран 9 не открылся

	(*10*) cmd_VS_Off := drm.cmd.9 := TRUE; //Останов воздушного стартера
	(*10*) drm.error.9 := am.KR13.notOff; //Кран 13 не закрылся

	(*11*) am.KR15.on := FALSE; //Кран 15 закрыть
	(*11*) drm.error.10 := am.KR15.notOff; //Кран 15 не закрылся

	(*12*) cmd_Kr4_Off := drm.cmd.11 := TRUE; //Кран 4 закрыть
	(*12*) drm.error.11 := am.Kr4.notOff; //Кран 4 не закрылся

	(*13*) cmd_KR11_Off := drm.cmd.12 := TRUE; //Закрытие крана 11, открытие крана 10

	(*14*) check_Nst := drm.cmd.13 := TRUE; //Проверка Nст
	(*14*) drm.error.13 := acpar.Nst.value > 100.0; //Nст > 100 об/мин

	//Условие перехода (1)→(2)
	//Кран 4 закрыт И Nст < 100 об/мин
	IF (am.Kr4.isOFF AND ( acpar.Nst.value < 100.0 OR acpar.Nst.flt )) AND drm.timeout THEN
		drm.cmd := drm.error := 0; drm.timer_pt := cycle; drm.inc := FALSE; drm.step := 2;
		cmd_M_K := FALSE; //Запуск последовательности "Переход М-К"
		sh_ms_off := FALSE; //Снятие защиты по маслосистеме ТК и СТ
		cmd_KPV15_On := FALSE; //Открыть КПВ 1, 5
		cmd_KPV234_On := FALSE; //Открыть КПВ 2, 3, 4
		cmd_sh_TG_Off := FALSE; //Снятие защиты по ТГ
		cmd_PNU_S_On := FALSE; //Включение маслонасосов смазки и уплотнения
		cmd_KR12_Off := FALSE; //Закрытие крана 12, открытие крана 9
		cmd_VS_Off := FALSE; //Останов воздушного стартера
		cmd_Kr4_Off := FALSE; //Кран 4 закрыть
		cmd_KR11_Off := FALSE; //Закрытие крана 11, открытие крана 10
		check_Nst := FALSE; //Проверка Nст
	END_IF;
2:	//Запись уставки таймера шага
	drm.step := 2;//Текущий шаг
	drm.timer_pt := cycle; //Таймер: один цикл вызова

	//Команды текущего шага
	(*1*) cmd_bleeding := drm.cmd.0 := drm.step_time <= cycle; //Запуск последовательности "Стравливание контура компрессора"

	//Условие перехода (2)→(3)
	//Подрежим "Стравливание контура компрессора" завершен
	IF (bleeding.finish) AND drm.timeout THEN
		drm.cmd := drm.error := 0; drm.timer_pt := cycle; drm.inc := FALSE; drm.step := 3;
		cmd_bleeding := FALSE; //Запуск последовательности "Стравливание контура компрессора"
	END_IF;
3:	//Запись уставки таймера шага
	drm.step := 3;//Текущий шаг
	drm.timer_pt := 60; //Таймер: 60 секунд

	//Команды текущего шага
	(*1*) check_Ntk := drm.cmd.0 := TRUE; //Выбег двигателя

	//Условие перехода (3)→(4)
	//Логическая 1
	IF (TRUE) AND drm.timeout THEN
		drm.cmd := drm.error := 0; drm.timer_pt := cycle; drm.inc := FALSE; drm.step := 4;
		check_Ntk := FALSE; //Выбег двигателя
	END_IF;
4:	//Запись уставки таймера шага
	drm.step := 4;//Текущий шаг
	drm.timer_pt := 2; //Таймер: 2 секунд

	//Команды текущего шага
	(*1*) cmd_VNA_On := FALSE; //Отключение Э/М ВНА

	(*2*) cmd_shPmN_Off := drm.cmd.1 := TRUE; //Снятие защиты по маслосистеме нагнетателя

	(*3*) cmd_sh_dPmg_Off := drm.cmd.2 := TRUE; //Снятие защиты по перепаду "масло-газ"

	//Условие перехода (4)→(5)
	//Логическая 1
	IF (TRUE) AND drm.timeout THEN
		drm.cmd := drm.error := 0; drm.timer_pt := cycle; drm.inc := FALSE; drm.step := 5;
		cmd_shPmN_Off := FALSE; //Снятие защиты по маслосистеме нагнетателя
		cmd_sh_dPmg_Off := FALSE; //Снятие защиты по перепаду "масло-газ"
	END_IF;
5:	//Запись уставки таймера шага
	drm.step := 5;//Текущий шаг
	drm.timer_pt := cycle; //Таймер: один цикл вызова

	//Команды текущего шага
	(*1*) cmd_PNU_S_Off := drm.cmd.0 := TRUE; //Пуск таймера отключения ПНС, ПНУ

	//Условие перехода (5)→(6)
	//Логическая 1
	IF (TRUE) AND drm.timeout THEN
		drm.cmd := drm.error := 0; drm.timer_pt := cycle; drm.inc := FALSE; drm.step := 6;
		cmd_PNU_S_Off := FALSE; //Пуск таймера отключения ПНС, ПНУ
	END_IF;
6:	//Запись уставки таймера шага
	drm.step := 6;//Текущий шаг
	drm.timer_pt := cycle; //Таймер: один цикл вызова

	//Команды текущего шага
	(*1*) finish := drm.cmd.0 := TRUE; //Завершение
	(*1*) drm.error.0 := NOT tch.Unlock.value; //АОсс завершен, нажмите кнопку "Деблокировка"

	//Условие перехода (6)→(0)
	//Деблокировка
	IF (tch.Unlock.value) AND drm.timeout THEN
		drm.cmd := drm.error := 0; drm.timer_pt := cycle; drm.inc := FALSE; drm.step := -1;
		finish := FALSE; //Завершение
	END_IF;
END_CASE

//Принудительный выход из последовательности
IF break THEN
	drm.step := -1; drm.cmd := drm.error := 0; drm.timer_pt := cycle; drm.inc := FALSE;
	emergStopCom := FALSE; //Аварийный останов двигателя
	cmd_M_K := FALSE; //Запуск последовательности "Переход М-К"
	sh_ms_off := FALSE; //Снятие защиты по маслосистеме ТК и СТ
	cmd_KPV15_On := FALSE; //Открыть КПВ 1, 5
	cmd_KPV234_On := FALSE; //Открыть КПВ 2, 3, 4
	cmd_VNA_On := FALSE; //Включение Э/М ВНА
	cmd_sh_TG_Off := FALSE; //Снятие защиты по ТГ
	cmd_PNU_S_On := FALSE; //Включение маслонасосов смазки и уплотнения
	cmd_KR12_Off := FALSE; //Закрытие крана 12, открытие крана 9
	cmd_VS_Off := FALSE; //Останов воздушного стартера
	cmd_Kr4_Off := FALSE; //Кран 4 закрыть
	cmd_KR11_Off := FALSE; //Закрытие крана 11, открытие крана 10
	check_Nst := FALSE; //Проверка Nст
	cmd_bleeding := FALSE; //Запуск последовательности "Стравливание контура компрессора"
	check_Ntk := FALSE; //Выбег двигателя
	cmd_shPmN_Off := FALSE; //Снятие защиты по маслосистеме нагнетателя
	cmd_sh_dPmg_Off := FALSE; //Снятие защиты по перепаду "масло-газ"
	cmd_PNU_S_Off := FALSE; //Пуск таймера отключения ПНС, ПНУ
	finish := FALSE; //Завершение
END_IF;

                  
END_FUNCTION_BLOCK

{region INFO}
(*
 Наименование последовательности: АПК
 Автор: /Разработчик/ 08.08.2025 9:04:03
 Версия: v00.00.18
 Проект: KA107
*)
{endregion}
{attribute 'symbol' := 'none'}
FUNCTION_BLOCK PUBLIC T_APK
VAR_INPUT
	cycle : REAL; //цикл вызова
END_VAR
VAR_OUTPUT
	cmd_sound_On : BOOL; //Предпусковая сигнализация
	cmd_PNU_S_On : BOOL; //Включение маслонасосов смазки и уплотнения
	cmd_shPmN_On : BOOL; //Взвод защиты по маслосистеме нагнетателя
	cmd_sh_dPmg_On : BOOL; //Взвод защиты по перепаду "масло-газ"
	cmd_filling : BOOL; //Запуск последовательности "Заполнение контура компрессора"
	cmd_start_D : BOOL; //Запуск последовательности "Пуск двигателя"
	finish : BOOL; //Завершение
	{attribute 'symbol' := 'read'}
	drm : Tdrm; //Интерфейсный функциональный блок
END_VAR
VAR
	start : BOOL; //Запуск последовательности
	break : BOOL; //Принудительный выход из последовательности
END_VAR

                    //Собираем переходы для визуализации
drm.transition.0 := start := mde.APK; //Запуск последовательности (0→1): Режим АПК
drm.transition.1 := TRUE; //1→2: Логическая 1
drm.transition.2 := aipar.dPmg.value > 0.5 AND NOT dipar.Pm_N_Pn.value; //2→3: dP масло-газ > 0.5 кгс/см2 и Pm > 1 кгс/см2
drm.transition.3 := Filling.finish; //3→4: Подсистема "Газовая обвязка" запущена
drm.transition.4 := FuelReg.fReg.started; //4→5: Двигатель перешел в режим "Работа"
drm.transition.5 := TRUE; //5→0: Логическая 1
drm.transition.31 := break := alg.AO; //Принудительный выход из последовательности (N→0): Режимы аварийного останова

//Вызываем экземпляр интерфейсного функционального блока
drm(cycle := cycle);

CASE drm.step OF
-1:	//Сброс команд с предыдущих шагов
	finish := FALSE;
	//Условие запуска последовательности
	//Режим АПК
	IF start AND NOT break THEN drm.step := 1; END_IF;
1:	//Запись уставки таймера шага
	drm.step := 1;//Текущий шаг
	drm.timer_pt := 10; //Таймер: 10 секунд

	//Команды текущего шага
	(*1*) cmd_sound_On := drm.cmd.0 := TRUE; //Предпусковая сигнализация

	//Условие перехода (1)→(2)
	//Логическая 1
	IF (TRUE) AND drm.timeout THEN
		drm.cmd := drm.error := 0; drm.timer_pt := cycle; drm.inc := FALSE; drm.step := 2;
		cmd_sound_On := FALSE; //Предпусковая сигнализация
	END_IF;
2:	//Запись уставки таймера шага
	drm.step := 2;//Текущий шаг
	drm.timer_pt := cycle; //Таймер: один цикл вызова

	//Команды текущего шага
	(*1*) cmd_PNU_S_On := drm.cmd.0 := TRUE; //Включение маслонасосов смазки и уплотнения

	//Условие перехода (2)→(3)
	//dP масло-газ > 0.5 кгс/см2 и Pm > 1 кгс/см2
	IF (aipar.dPmg.value > 0.5 AND NOT dipar.Pm_N_Pn.value) AND drm.timeout THEN
		drm.cmd := drm.error := 0; drm.timer_pt := cycle; drm.inc := FALSE; drm.step := 3;
		cmd_PNU_S_On := FALSE; //Включение маслонасосов смазки и уплотнения
	END_IF;
3:	//Запись уставки таймера шага
	drm.step := 3;//Текущий шаг
	drm.timer_pt := cycle; //Таймер: один цикл вызова

	//Команды текущего шага
	(*1*) cmd_shPmN_On := drm.cmd.0 := TRUE; //Взвод защиты по маслосистеме нагнетателя

	(*2*) cmd_sh_dPmg_On := drm.cmd.1 := TRUE; //Взвод защиты по перепаду "масло-газ"

	(*3*) cmd_filling := drm.cmd.2 := drm.step_time <= cycle; //Запуск последовательности "Заполнение контура компрессора"

	//Условие перехода (3)→(4)
	//Подсистема "Газовая обвязка" запущена
	IF (Filling.finish) AND drm.timeout THEN
		drm.cmd := drm.error := 0; drm.timer_pt := cycle; drm.inc := FALSE; drm.step := 4;
		cmd_shPmN_On := FALSE; //Взвод защиты по маслосистеме нагнетателя
		cmd_sh_dPmg_On := FALSE; //Взвод защиты по перепаду "масло-газ"
		cmd_filling := FALSE; //Запуск последовательности "Заполнение контура компрессора"
	END_IF;
4:	//Запись уставки таймера шага
	drm.step := 4;//Текущий шаг
	drm.inc := TRUE; //Выставляем признак инкремента

	//Команды текущего шага
	(*1*) cmd_start_D := drm.cmd.0 := drm.step_time <= cycle; //Запуск последовательности "Пуск двигателя"

	//Условие перехода (4)→(5)
	//Двигатель перешел в режим "Работа"
	IF (FuelReg.fReg.started) AND drm.timeout THEN
		drm.cmd := drm.error := 0; drm.timer_pt := cycle; drm.inc := FALSE; drm.step := 5;
		cmd_start_D := FALSE; //Запуск последовательности "Пуск двигателя"
	END_IF;
5:	//Запись уставки таймера шага
	drm.step := 5;//Текущий шаг
	drm.timer_pt := cycle; //Таймер: один цикл вызова

	//Команды текущего шага
	(*1*) finish := drm.cmd.0 := TRUE; //Завершение

	//Условие перехода (5)→(0)
	//Логическая 1
	IF (TRUE) AND drm.timeout THEN
		drm.cmd := drm.error := 0; drm.timer_pt := cycle; drm.inc := FALSE; drm.step := -1;
		finish := FALSE; //Завершение
	END_IF;
END_CASE

//Принудительный выход из последовательности
IF break THEN
	drm.step := -1; drm.cmd := drm.error := 0; drm.timer_pt := cycle; drm.inc := FALSE;
	cmd_sound_On := FALSE; //Предпусковая сигнализация
	cmd_PNU_S_On := FALSE; //Включение маслонасосов смазки и уплотнения
	cmd_shPmN_On := FALSE; //Взвод защиты по маслосистеме нагнетателя
	cmd_sh_dPmg_On := FALSE; //Взвод защиты по перепаду "масло-газ"
	cmd_filling := FALSE; //Запуск последовательности "Заполнение контура компрессора"
	cmd_start_D := FALSE; //Запуск последовательности "Пуск двигателя"
	finish := FALSE; //Завершение
END_IF;

                  
END_FUNCTION_BLOCK

{region INFO}
(*
 Наименование последовательности: Стравливание
 Автор: /Разработчик/ 08.08.2025 9:04:03
 Версия: v00.00.18
 Проект: KA107
*)
{endregion}
{attribute 'symbol' := 'none'}
FUNCTION_BLOCK PUBLIC T_Bleeding_full
VAR_INPUT
	cycle : REAL; //цикл вызова
END_VAR
VAR_OUTPUT
	cmd_bleeding : BOOL; //Запуск последовательности "Стравливание контура компрессора"
	cmd_sh_dPmg_Off : BOOL; //Снятие защиты по перепаду "масло-газ"
	cmd_shPmN_Off : BOOL; //Снятие защиты по маслосистеме нагнетателя
	cmd_PNU_S_Off : BOOL; //Пуск таймера отключения ПНС, ПНУ
	finish : BOOL; //Завершение
	{attribute 'symbol' := 'read'}
	drm : Tdrm; //Интерфейсный функциональный блок
END_VAR
VAR
	start : BOOL; //Запуск последовательности
	break : BOOL; //Принудительный выход из последовательности
END_VAR

                    //Собираем переходы для визуализации
drm.transition.0 := start := btn.Bleeding.out; //Запуск последовательности (0→1): Нажата кнопка "Стравливание"
drm.transition.1 := bleeding.finish; //1→2: Подрежим "Стравливание контура компрессора" завершен
drm.transition.2 := TRUE; //2→3: Логическая 1
drm.transition.3 := TRUE; //3→0: Логическая 1
drm.transition.31 := break := mde.AOss; //Принудительный выход из последовательности (N→0): Режим АОсс

//Вызываем экземпляр интерфейсного функционального блока
drm(cycle := cycle);

CASE drm.step OF
-1:	//Сброс команд с предыдущих шагов
	finish := FALSE;
	//Условие запуска последовательности
	//Нажата кнопка "Стравливание"
	IF start AND NOT break THEN drm.step := 1; END_IF;
1:	//Запись уставки таймера шага
	drm.step := 1;//Текущий шаг
	drm.timer_pt := cycle; //Таймер: один цикл вызова

	//Команды текущего шага
	(*1*) cmd_bleeding := drm.cmd.0 := drm.step_time <= cycle; //Запуск последовательности "Стравливание контура компрессора"

	//Условие перехода (1)→(2)
	//Подрежим "Стравливание контура компрессора" завершен
	IF (bleeding.finish) AND drm.timeout THEN
		drm.cmd := drm.error := 0; drm.timer_pt := cycle; drm.inc := FALSE; drm.step := 2;
		cmd_bleeding := FALSE; //Запуск последовательности "Стравливание контура компрессора"
	END_IF;
2:	//Запись уставки таймера шага
	drm.step := 2;//Текущий шаг
	drm.timer_pt := cycle; //Таймер: один цикл вызова

	//Команды текущего шага
	(*1*) cmd_sh_dPmg_Off := drm.cmd.0 := TRUE; //Снятие защиты по перепаду "масло-газ"

	(*2*) cmd_shPmN_Off := drm.cmd.1 := TRUE; //Снятие защиты по маслосистеме нагнетателя

	(*3*) cmd_PNU_S_Off := drm.cmd.2 := TRUE; //Пуск таймера отключения ПНС, ПНУ

	//Условие перехода (2)→(3)
	//Логическая 1
	IF (TRUE) AND drm.timeout THEN
		drm.cmd := drm.error := 0; drm.timer_pt := cycle; drm.inc := FALSE; drm.step := 3;
		cmd_sh_dPmg_Off := FALSE; //Снятие защиты по перепаду "масло-газ"
		cmd_shPmN_Off := FALSE; //Снятие защиты по маслосистеме нагнетателя
		cmd_PNU_S_Off := FALSE; //Пуск таймера отключения ПНС, ПНУ
	END_IF;
3:	//Запись уставки таймера шага
	drm.step := 3;//Текущий шаг
	drm.timer_pt := cycle; //Таймер: один цикл вызова

	//Команды текущего шага
	(*1*) finish := drm.cmd.0 := TRUE; //Завершение

	//Условие перехода (3)→(0)
	//Логическая 1
	IF (TRUE) AND drm.timeout THEN
		drm.cmd := drm.error := 0; drm.timer_pt := cycle; drm.inc := FALSE; drm.step := -1;
		finish := FALSE; //Завершение
	END_IF;
END_CASE

//Принудительный выход из последовательности
IF break THEN
	drm.step := -1; drm.cmd := drm.error := 0; drm.timer_pt := cycle; drm.inc := FALSE;
	cmd_bleeding := FALSE; //Запуск последовательности "Стравливание контура компрессора"
	cmd_sh_dPmg_Off := FALSE; //Снятие защиты по перепаду "масло-газ"
	cmd_shPmN_Off := FALSE; //Снятие защиты по маслосистеме нагнетателя
	cmd_PNU_S_Off := FALSE; //Пуск таймера отключения ПНС, ПНУ
	finish := FALSE; //Завершение
END_IF;

                  
END_FUNCTION_BLOCK

{region INFO}
(*
 Наименование последовательности: Контроль САУ
 Автор: /Разработчик/ 08.08.2025 9:04:03
 Версия: v00.00.18
 Проект: KA107
*)
{endregion}
{attribute 'symbol' := 'none'}
FUNCTION_BLOCK PUBLIC T_Check_SAU
VAR_INPUT
	cycle : REAL; //цикл вызова
END_VAR
VAR_OUTPUT
	cmd_check_VibD : BOOL; //Контроль виброаппаратуры двигателя
	cmd_check_BZA : BOOL; //Контроль БЗА двигателя
	wait_crs : BOOL; //Ожидание аварийных сигнализаций
	finish : BOOL; //Завершение
	{attribute 'symbol' := 'read'}
	drm : Tdrm; //Интерфейсный функциональный блок
END_VAR
VAR
	start : BOOL; //Запуск последовательности
	break : BOOL; //Принудительный выход из последовательности
END_VAR

                    //Собираем переходы для визуализации
drm.transition.0 := start := check.btn OR btn.Check_SAU.out OR check.tmr12H.Q; //Запуск последовательности (0→1): Нажата одна из пусковых кнопок ИЛИ Кнопка "Контроль САУ" ИЛИ Каждые 12 часов
drm.transition.1 := crs.Vs_D_Av.signalization AND crs.BZA_alr.signalization AND crs.Vsst_HH.signalization AND crs.Vstk_HH.signalization; //1→2: Сформированы аварийные сигнализации двигателя
drm.transition.2 := TRUE; //2→0: Логическая 1
drm.transition.31 := break := btn.Cancel.out; //Принудительный выход из последовательности (N→0): Деблокировка

//Вызываем экземпляр интерфейсного функционального блока
drm(cycle := cycle);

CASE drm.step OF
-1:	//Сброс команд с предыдущих шагов
	finish := FALSE;
	//Условие запуска последовательности
	//Нажата одна из пусковых кнопок ИЛИ Кнопка "Контроль САУ" ИЛИ Каждые 12 часов
	IF start AND NOT break THEN drm.step := 1; END_IF;
1:	//Запись уставки таймера шага
	drm.step := 1;//Текущий шаг
	drm.timer_pt := 10; //Таймер: 10 секунд

	//Команды текущего шага
	(*1*) cmd_check_VibD := drm.cmd.0 := TRUE; //Контроль виброаппаратуры двигателя

	(*2*) cmd_check_BZA := drm.cmd.1 := TRUE; //Контроль БЗА двигателя

	(*3*) wait_crs := drm.cmd.2 := TRUE; //Ожидание аварийных сигнализаций

	//Условие перехода (1)→(2)
	//Сформированы аварийные сигнализации двигателя
	IF (crs.Vs_D_Av.signalization AND crs.BZA_alr.signalization AND crs.Vsst_HH.signalization AND crs.Vstk_HH.signalization) AND drm.timeout THEN
		drm.cmd := drm.error := 0; drm.timer_pt := cycle; drm.inc := FALSE; drm.step := 2;
		cmd_check_VibD := FALSE; //Контроль виброаппаратуры двигателя
		cmd_check_BZA := FALSE; //Контроль БЗА двигателя
		wait_crs := FALSE; //Ожидание аварийных сигнализаций
	END_IF;
2:	//Запись уставки таймера шага
	drm.step := 2;//Текущий шаг
	drm.timer_pt := cycle; //Таймер: один цикл вызова

	//Команды текущего шага
	(*1*) finish := drm.cmd.0 := TRUE; //Завершение

	//Условие перехода (2)→(0)
	//Логическая 1
	IF (TRUE) AND drm.timeout THEN
		drm.cmd := drm.error := 0; drm.timer_pt := cycle; drm.inc := FALSE; drm.step := -1;
		finish := FALSE; //Завершение
	END_IF;
END_CASE

//Принудительный выход из последовательности
IF break THEN
	drm.step := -1; drm.cmd := drm.error := 0; drm.timer_pt := cycle; drm.inc := FALSE;
	cmd_check_VibD := FALSE; //Контроль виброаппаратуры двигателя
	cmd_check_BZA := FALSE; //Контроль БЗА двигателя
	wait_crs := FALSE; //Ожидание аварийных сигнализаций
	finish := FALSE; //Завершение
END_IF;

                  
END_FUNCTION_BLOCK

{region INFO}
(*
 Наименование последовательности: ХП
 Автор: /Разработчик/ 08.08.2025 9:04:03
 Версия: v00.00.18
 Проект: KA107
*)
{endregion}
{attribute 'symbol' := 'none'}
FUNCTION_BLOCK PUBLIC T_HP
VAR_INPUT
	cycle : REAL; //цикл вызова
END_VAR
VAR_OUTPUT
	cmd_sound_On : BOOL; //Предпусковая сигнализация
	cmd_PNU_S_On : BOOL; //Пуск маслонасосов смазки и уплотнения
	cmd_shPmN_On : BOOL; //Взвод защиты по маслосистеме нагнетателя
	cmd_sh_dPmg_On : BOOL; //Взвод защиты по перепаду "масло-газ"
	cmd_KR11_On : BOOL; //Открытие крана 11, закрытие крана 10
	check : BOOL; //Проверка Nвд
	cmd_VS_On : BOOL; //Пуск воздушного стартера
	cmd_sh_Pm_Starter : BOOL; //Взвод защиты по давлению масла ВС
	cmd_HP_D : BOOL; //Холодная прокрутка двигателя
	cmd_VS_Off : BOOL; //Останов воздушного стартера
	cmd_KR11_Off : BOOL; //Закрытие крана 11, открытие крана 10
	cmd_HP_stop_D : BOOL; //Выбег двигателя после ХП
	cmd_shPmN_Off : BOOL; //Снятие защиты по маслосистеме
	cmd_PNU_Off : BOOL; //Отключение маслонасоса уплотнения
	cmd_sh_dPmg_Off : BOOL; //Снятие защиты по перепаду "масло-газ"
	cmd_PNS_Off : BOOL; //Отключение маслонасоса смазки
	finish : BOOL; //Завершение
	{attribute 'symbol' := 'read'}
	drm : Tdrm; //Интерфейсный функциональный блок
END_VAR
VAR
	start : BOOL; //Запуск последовательности
	break : BOOL; //Принудительный выход из последовательности
END_VAR

                    //Собираем переходы для визуализации
drm.transition.0 := start := mde.HP; //Запуск последовательности (0→1): Режим ХП
drm.transition.1 := TRUE; //1→2: Логическая 1
drm.transition.2 := aipar.dPmg.value > 0.5 AND NOT dipar.Pm_N_Pn.value; //2→3: dP масло-газ > 0.5 кгс/см2 и Pm > 1 кгс/см2
drm.transition.3 := am.KR11.isOn AND am.KR10.isOff; //3→4: Кран 11 открылся, кран 10 закрылся
drm.transition.4 := acpar.Ntk.value < 100.0; //4→5: Nвд < 100 об/мин
drm.transition.5 := TRUE; //5→6: Логическая 1
drm.transition.6 := TRUE; //6→7: Логическая 1
drm.transition.7 := am.KR13.isOff; //7→8: Холодная прокрутка двигателя завершена
drm.transition.8 := acpar.Ntk.value < 100 AND tch.nGas_N.value; //8→9: Nтк < 100 И Нет газа в контуре
drm.transition.9 := acpar.Ntk.value < 100 AND tch.Gas_N.value; //8→11: Nтк < 100 И Есть газ в контуре
drm.transition.10 := TRUE; //9→10: Логическая 1
drm.transition.11 := TRUE; //10→11: Логическая 1
drm.transition.12 := TRUE; //11→0: Логическая 1
drm.transition.31 := break := NOT mde.HP; //Принудительный выход из последовательности (N→0): Снятие режима

//Вызываем экземпляр интерфейсного функционального блока
drm(cycle := cycle);

CASE drm.step OF
-1:	//Сброс команд с предыдущих шагов
	finish := FALSE;
	//Условие запуска последовательности
	//Режим ХП
	IF start AND NOT break THEN drm.step := 1; END_IF;
1:	//Запись уставки таймера шага
	drm.step := 1;//Текущий шаг
	drm.timer_pt := 10; //Таймер: 10 секунд

	//Команды текущего шага
	(*1*) cmd_sound_On := drm.cmd.0 := TRUE; //Предпусковая сигнализация

	//Условие перехода (1)→(2)
	//Логическая 1
	IF (TRUE) AND drm.timeout THEN
		drm.cmd := drm.error := 0; drm.timer_pt := cycle; drm.inc := FALSE; drm.step := 2;
		cmd_sound_On := FALSE; //Предпусковая сигнализация
	END_IF;
2:	//Запись уставки таймера шага
	drm.step := 2;//Текущий шаг
	drm.timer_pt := cycle; //Таймер: один цикл вызова

	//Команды текущего шага
	(*1*) cmd_PNU_S_On := drm.cmd.0 := TRUE; //Пуск маслонасосов смазки и уплотнения

	//Условие перехода (2)→(3)
	//dP масло-газ > 0.5 кгс/см2 и Pm > 1 кгс/см2
	IF (aipar.dPmg.value > 0.5 AND NOT dipar.Pm_N_Pn.value) AND drm.timeout THEN
		drm.cmd := drm.error := 0; drm.timer_pt := cycle; drm.inc := FALSE; drm.step := 3;
		cmd_PNU_S_On := FALSE; //Пуск маслонасосов смазки и уплотнения
	END_IF;
3:	//Запись уставки таймера шага
	drm.step := 3;//Текущий шаг
	drm.timer_pt := cycle; //Таймер: один цикл вызова

	//Команды текущего шага
	(*1*) cmd_shPmN_On := drm.cmd.0 := TRUE; //Взвод защиты по маслосистеме нагнетателя

	(*2*) cmd_sh_dPmg_On := drm.cmd.1 := TRUE; //Взвод защиты по перепаду "масло-газ"

	(*3*) cmd_KR11_On := drm.cmd.2 := TRUE; //Открытие крана 11, закрытие крана 10
	(*3*) drm.error.2 := am.KR11.notOn OR am.KR10.notOff; //Кран 11 не открылся, кран 10 не закрылся

	//Условие перехода (3)→(4)
	//Кран 11 открылся, кран 10 закрылся
	IF (am.KR11.isOn AND am.KR10.isOff) AND drm.timeout THEN
		drm.cmd := drm.error := 0; drm.timer_pt := cycle; drm.inc := FALSE; drm.step := 4;
		cmd_shPmN_On := FALSE; //Взвод защиты по маслосистеме нагнетателя
		cmd_sh_dPmg_On := FALSE; //Взвод защиты по перепаду "масло-газ"
		cmd_KR11_On := FALSE; //Открытие крана 11, закрытие крана 10
	END_IF;
4:	//Запись уставки таймера шага
	drm.step := 4;//Текущий шаг
	drm.timer_pt := cycle; //Таймер: один цикл вызова

	//Команды текущего шага
	(*1*) check := drm.cmd.0 := TRUE; //Проверка Nвд
	(*1*) drm.error.0 := acpar.Ntk.value > 100.0; //Nвд > 100 об/мин

	//Условие перехода (4)→(5)
	//Nвд < 100 об/мин
	IF (acpar.Ntk.value < 100.0) AND drm.timeout THEN
		drm.cmd := drm.error := 0; drm.timer_pt := cycle; drm.inc := FALSE; drm.step := 5;
		check := FALSE; //Проверка Nвд
	END_IF;
5:	//Запись уставки таймера шага
	drm.step := 5;//Текущий шаг
	drm.timer_pt := cycle; //Таймер: один цикл вызова

	//Команды текущего шага
	(*1*) cmd_VS_On := drm.cmd.0 := drm.step_time <= cycle; //Пуск воздушного стартера
	(*1*) drm.error.0 := am.KR13.notOn; //Кран 13 не открылся

	//Условие перехода (5)→(6)
	//Логическая 1
	IF (TRUE) AND drm.timeout THEN
		drm.cmd := drm.error := 0; drm.timer_pt := cycle; drm.inc := FALSE; drm.step := 6;
		cmd_VS_On := FALSE; //Пуск воздушного стартера
	END_IF;
6:	//Запись уставки таймера шага
	drm.step := 6;//Текущий шаг
	drm.timer_pt := 120; //Таймер: 120 секунд

	//Команды текущего шага
	(*1*) cmd_sh_Pm_Starter := drm.cmd.0 := drm.step_time <= cycle; //Взвод защиты по давлению масла ВС

	(*2*) cmd_HP_D := drm.cmd.1 := drm.step_time <= cycle; //Холодная прокрутка двигателя

	//Условие перехода (6)→(7)
	//Логическая 1
	IF (TRUE) AND drm.timeout THEN
		drm.cmd := drm.error := 0; drm.timer_pt := cycle; drm.inc := FALSE; drm.step := 7;
		cmd_sh_Pm_Starter := FALSE; //Взвод защиты по давлению масла ВС
		cmd_HP_D := FALSE; //Холодная прокрутка двигателя
	END_IF;
7:	//Запись уставки таймера шага
	drm.step := 7;//Текущий шаг
	drm.timer_pt := cycle; //Таймер: один цикл вызова

	//Команды текущего шага
	(*1*) cmd_VS_Off := drm.cmd.0 := TRUE; //Останов воздушного стартера
	(*1*) drm.error.0 := am.KR13.notOff; //Кран 13 не закрылся

	//Условие перехода (7)→(8)
	//Холодная прокрутка двигателя завершена
	IF (am.KR13.isOff) AND drm.timeout THEN
		drm.cmd := drm.error := 0; drm.timer_pt := cycle; drm.inc := FALSE; drm.step := 8;
		cmd_VS_Off := FALSE; //Останов воздушного стартера
	END_IF;
8:	//Запись уставки таймера шага
	drm.step := 8;//Текущий шаг
	drm.timer_pt := cycle; //Таймер: один цикл вызова

	//Команды текущего шага
	(*1*) cmd_KR11_Off := drm.cmd.0 := TRUE; //Закрытие крана 11, открытие крана 10
	(*1*) drm.error.0 := am.KR11.notOff OR am.KR10.notOn; //Кран 11 не закрылся, кран 10 не открылся

	(*2*) cmd_HP_stop_D := drm.cmd.1 := TRUE; //Выбег двигателя после ХП

	//Условие перехода на шаг (9)
	//Nтк < 100 И Нет газа в контуре
	IF (acpar.Ntk.value < 100 AND tch.nGas_N.value) AND drm.timeout THEN
		drm.cmd := drm.error := 0; drm.timer_pt := cycle; drm.inc := FALSE; drm.step := 9;
		cmd_KR11_Off := FALSE; //Закрытие крана 11, открытие крана 10
		cmd_HP_stop_D := FALSE; //Выбег двигателя после ХП
	END_IF;
	//Условие перехода (8)→(11)
	//Nтк < 100 И Есть газ в контуре
	IF (acpar.Ntk.value < 100 AND tch.Gas_N.value) AND drm.timeout THEN
		drm.cmd := drm.error := 0; drm.timer_pt := cycle; drm.inc := FALSE; drm.step := 11;
		cmd_KR11_Off := FALSE; //Закрытие крана 11, открытие крана 10
		cmd_HP_stop_D := FALSE; //Выбег двигателя после ХП
	END_IF;
9:	//Запись уставки таймера шага
	drm.step := 9;//Текущий шаг
	drm.timer_pt := 2; //Таймер: 2 секунд

	//Команды текущего шага
	(*1*) cmd_shPmN_Off := drm.cmd.0 := TRUE; //Снятие защиты по маслосистеме

	(*2*) cmd_PNU_Off := drm.cmd.1 := TRUE; //Отключение маслонасоса уплотнения
	(*2*) drm.error.1 := am.PNU.notOff; //Маслонасос уплотнений не выключился

	(*3*) cmd_sh_dPmg_Off := drm.cmd.2 := TRUE; //Снятие защиты по перепаду "масло-газ"

	//Условие перехода (9)→(10)
	//Логическая 1
	IF (TRUE) AND drm.timeout THEN
		drm.cmd := drm.error := 0; drm.timer_pt := cycle; drm.inc := FALSE; drm.step := 10;
		cmd_shPmN_Off := FALSE; //Снятие защиты по маслосистеме
		cmd_PNU_Off := FALSE; //Отключение маслонасоса уплотнения
		cmd_sh_dPmg_Off := FALSE; //Снятие защиты по перепаду "масло-газ"
	END_IF;
10:	//Запись уставки таймера шага
	drm.step := 10;//Текущий шаг
	drm.timer_pt := cycle; //Таймер: один цикл вызова

	//Команды текущего шага
	(*1*) cmd_PNS_Off := drm.cmd.0 := TRUE; //Отключение маслонасоса смазки
	(*1*) drm.error.0 := am.PNS.notOff; //Маслонасос смазки не выключился

	//Условие перехода (10)→(11)
	//Логическая 1
	IF (TRUE) AND drm.timeout THEN
		drm.cmd := drm.error := 0; drm.timer_pt := cycle; drm.inc := FALSE; drm.step := 11;
		cmd_PNS_Off := FALSE; //Отключение маслонасоса смазки
	END_IF;
11:	//Запись уставки таймера шага
	drm.step := 11;//Текущий шаг
	drm.timer_pt := cycle; //Таймер: один цикл вызова

	//Команды текущего шага
	(*1*) finish := drm.cmd.0 := drm.step_time <= cycle; //Завершение

	//Условие перехода (11)→(0)
	//Логическая 1
	IF (TRUE) AND drm.timeout THEN
		drm.cmd := drm.error := 0; drm.timer_pt := cycle; drm.inc := FALSE; drm.step := -1;
		finish := FALSE; //Завершение
	END_IF;
END_CASE

//Принудительный выход из последовательности
IF break THEN
	drm.step := -1; drm.cmd := drm.error := 0; drm.timer_pt := cycle; drm.inc := FALSE;
	cmd_sound_On := FALSE; //Предпусковая сигнализация
	cmd_PNU_S_On := FALSE; //Пуск маслонасосов смазки и уплотнения
	cmd_shPmN_On := FALSE; //Взвод защиты по маслосистеме нагнетателя
	cmd_sh_dPmg_On := FALSE; //Взвод защиты по перепаду "масло-газ"
	cmd_KR11_On := FALSE; //Открытие крана 11, закрытие крана 10
	check := FALSE; //Проверка Nвд
	cmd_VS_On := FALSE; //Пуск воздушного стартера
	cmd_sh_Pm_Starter := FALSE; //Взвод защиты по давлению масла ВС
	cmd_HP_D := FALSE; //Холодная прокрутка двигателя
	cmd_VS_Off := FALSE; //Останов воздушного стартера
	cmd_KR11_Off := FALSE; //Закрытие крана 11, открытие крана 10
	cmd_HP_stop_D := FALSE; //Выбег двигателя после ХП
	cmd_shPmN_Off := FALSE; //Снятие защиты по маслосистеме
	cmd_PNU_Off := FALSE; //Отключение маслонасоса уплотнения
	cmd_sh_dPmg_Off := FALSE; //Снятие защиты по перепаду "масло-газ"
	cmd_PNS_Off := FALSE; //Отключение маслонасоса смазки
	finish := FALSE; //Завершение
END_IF;

                  
END_FUNCTION_BLOCK

{region INFO}
(*
 Наименование последовательности: КПК
 Автор: /Разработчик/ 08.08.2025 9:04:03
 Версия: v00.00.18
 Проект: KA107
*)
{endregion}
{attribute 'symbol' := 'none'}
FUNCTION_BLOCK PUBLIC T_KPK
VAR_INPUT
	cycle : REAL; //цикл вызова
END_VAR
VAR_OUTPUT
	cmd_sound_On : BOOL; //Предпусковая сигнализация
	cmd_PNU_S_On : BOOL; //Пуск маслонасосов уплотнения и смазки
	cmd_sh_dPmg_On : BOOL; //Взвод защиты по перепаду "масло-газ"
	cmd_shPmN_On : BOOL; //Взвод защиты по маслосистеме нагнетателя
	cmd_filling : BOOL; //Запуск последовательности "Заполнение контура компрессора"
	cmd_KR12_On : BOOL; //Открытие крана 12, закрытие крана 9
	cmd_KR12_Off : BOOL; //Закрытие крана 12, открытие крана 9
	cmd_Kr6_Off : BOOL; //Кран 6 закрыть
	cmd_Kr1_Off : BOOL; //Кран 1 закрыть
	cmd_Kr2_Off : BOOL; //Кран 2 закрыть
	cmd_Kr4_On : BOOL; //Кран 4 открыть
	finish : BOOL; //Завершение
	{attribute 'symbol' := 'read'}
	drm : Tdrm; //Интерфейсный функциональный блок
END_VAR
VAR
	start : BOOL; //Запуск последовательности
	break : BOOL; //Принудительный выход из последовательности
END_VAR

                    //Собираем переходы для визуализации
drm.transition.0 := start := mde.KPK; //Запуск последовательности (0→1): Режим КПК
drm.transition.1 := TRUE; //1→2: Логическая 1
drm.transition.2 := aipar.dPmg.value > 0.5 AND NOT dipar.Pm_N_Pn.value; //2→3: dP масло-газ > 0.5 кгс/см2 и Pm > 1 кгс/см2
drm.transition.3 := subsystem.go.work; //3→4: Подсистема "Газовая обвязка" запущена
drm.transition.4 := am.KR12.isON AND am.KR9.isOff AND aipar.Ptg_inTRK.value > 1.96; //4→5: Кран 12 открылся И кран 9 закрылся И Pтг > 1.96
drm.transition.5 := am.KR12.isOFF AND am.KR9.isON; //5→6: Кран 12 закрылся И кран 9 открылся
drm.transition.6 := am.Kr6.isOFF; //6→7: Кран 6 закрыт
drm.transition.7 := am.Kr1.isOFF AND am.Kr2.isOFF AND am.Kr4.isON; //7→8: Кран 1 закрыт И Кран 2 закрыт И Кран 4 открыт
drm.transition.8 := TRUE; //8→0: Логическая 1
drm.transition.31 := break := NOT mde.KPK; //Принудительный выход из последовательности (N→0): Снятие режима

//Вызываем экземпляр интерфейсного функционального блока
drm(cycle := cycle);

CASE drm.step OF
-1:	//Сброс команд с предыдущих шагов
	finish := FALSE;
	//Условие запуска последовательности
	//Режим КПК
	IF start AND NOT break THEN drm.step := 1; END_IF;
1:	//Запись уставки таймера шага
	drm.step := 1;//Текущий шаг
	drm.timer_pt := 10; //Таймер: 10 секунд

	//Команды текущего шага
	(*1*) cmd_sound_On := drm.cmd.0 := TRUE; //Предпусковая сигнализация

	//Условие перехода (1)→(2)
	//Логическая 1
	IF (TRUE) AND drm.timeout THEN
		drm.cmd := drm.error := 0; drm.timer_pt := cycle; drm.inc := FALSE; drm.step := 2;
		cmd_sound_On := FALSE; //Предпусковая сигнализация
	END_IF;
2:	//Запись уставки таймера шага
	drm.step := 2;//Текущий шаг
	drm.timer_pt := cycle; //Таймер: один цикл вызова

	//Команды текущего шага
	(*1*) cmd_PNU_S_On := drm.cmd.0 := TRUE; //Пуск маслонасосов уплотнения и смазки
	(*1*) drm.error.0 := am.PNU.notOn; //Маслонасос уплотнений не включился

	//Условие перехода (2)→(3)
	//dP масло-газ > 0.5 кгс/см2 и Pm > 1 кгс/см2
	IF (aipar.dPmg.value > 0.5 AND NOT dipar.Pm_N_Pn.value) AND drm.timeout THEN
		drm.cmd := drm.error := 0; drm.timer_pt := cycle; drm.inc := FALSE; drm.step := 3;
		cmd_PNU_S_On := FALSE; //Пуск маслонасосов уплотнения и смазки
	END_IF;
3:	//Запись уставки таймера шага
	drm.step := 3;//Текущий шаг
	drm.timer_pt := cycle; //Таймер: один цикл вызова

	//Команды текущего шага
	(*1*) cmd_sh_dPmg_On := drm.cmd.0 := TRUE; //Взвод защиты по перепаду "масло-газ"

	(*2*) cmd_shPmN_On := drm.cmd.1 := TRUE; //Взвод защиты по маслосистеме нагнетателя

	(*3*) cmd_filling := drm.cmd.2 := drm.step_time <= cycle; //Запуск последовательности "Заполнение контура компрессора"

	//Условие перехода (3)→(4)
	//Подсистема "Газовая обвязка" запущена
	IF (subsystem.go.work) AND drm.timeout THEN
		drm.cmd := drm.error := 0; drm.timer_pt := cycle; drm.inc := FALSE; drm.step := 4;
		cmd_sh_dPmg_On := FALSE; //Взвод защиты по перепаду "масло-газ"
		cmd_shPmN_On := FALSE; //Взвод защиты по маслосистеме нагнетателя
		cmd_filling := FALSE; //Запуск последовательности "Заполнение контура компрессора"
	END_IF;
4:	//Запись уставки таймера шага
	drm.step := 4;//Текущий шаг
	drm.timer_pt := cycle; //Таймер: один цикл вызова

	//Команды текущего шага
	(*1*) cmd_KR12_On := drm.cmd.0 := TRUE; //Открытие крана 12, закрытие крана 9
	(*1*) drm.error.0 := am.KR12.notOn OR am.KR9.notOff; //Кран 12 не открылся, кран 9 не закрылся

	//Условие перехода (4)→(5)
	//Кран 12 открылся И кран 9 закрылся И Pтг > 1.96
	IF (am.KR12.isON AND am.KR9.isOff AND aipar.Ptg_inTRK.value > 1.96) AND drm.timeout THEN
		drm.cmd := drm.error := 0; drm.timer_pt := cycle; drm.inc := FALSE; drm.step := 5;
		cmd_KR12_On := FALSE; //Открытие крана 12, закрытие крана 9
	END_IF;
5:	//Запись уставки таймера шага
	drm.step := 5;//Текущий шаг
	drm.timer_pt := cycle; //Таймер: один цикл вызова

